LIN {X 0,Y 573.259,Z 217.079,A -85,B 0,C 180,E1 -2322.989,E2 -2322.989} C_VEL
LIN {X 0,Y 573.272,Z 217.08,A -85,B 0,C 180,E1 -2325.806,E2 -2325.806} C_VEL
LIN {X 0,Y 573.26,Z 217.081,A -85,B 0,C 180,E1 -2328.744,E2 -2328.744} C_VEL
LIN {X 0,Y 573.283,Z 217.076,A -85,B 0,C 180,E1 -2331.539,E2 -2331.539} C_VEL
LIN {X 0,Y 573.295,Z 217.075,A -85,B 0,C 180,E1 -2334.371,E2 -2334.371} C_VEL
LIN {X 0,Y 573.306,Z 217.073,A -85,B 0,C 180,E1 -2337.891,E2 -2337.891} C_VEL
LIN {X 0,Y 573.333,Z 217.07,A -85,B 0,C 180,E1 -2340.701,E2 -2340.701} C_VEL
LIN {X 0,Y 573.233,Z 217.085,A -85,B 0,C 180,E1 -2343.513,E2 -2343.513} C_VEL
LIN {X 0,Y 573.286,Z 217.078,A -85,B 0,C 180,E1 -2345.627,E2 -2345.627} C_VEL
LIN {X 0,Y 573.304,Z 217.075,A -85,B 0,C 180,E1 -2348.458,E2 -2348.458} C_VEL
LIN {X 0,Y 573.238,Z 217.083,A -85,B 0,C 180,E1 -2351.311,E2 -2351.311} C_VEL
LIN {X 0,Y 573.113,Z 217.279,A -85,B 0,C 180,E1 -2352.751,E2 -2352.751} C_VEL
LIN {X 0,Y 573.098,Z 219.875,A -85,B 0,C 180,E1 -2354.922,E2 -2354.922} C_VEL
LIN {X 0,Y 573.095,Z 222.437,A -85,B 0,C 180,E1 -2357.115,E2 -2357.115} C_VEL
LIN {X 0,Y 573.071,Z 224.992,A -85,B 0,C 180,E1 -2359.335,E2 -2359.335} C_VEL
LIN {X 0,Y 573.008,Z 227.552,A -85,B 0,C 180,E1 -2361.588,E2 -2361.588} C_VEL
LIN {X 0,Y 572.988,Z 230.552,A -85,B 0,C 180,E1 -2364.29,E2 -2364.29} C_VEL
LIN {X 0,Y 572.316,Z 231.276,A -85,B 0,C 180,E1 -2364.872,E2 -2364.872} C_VEL
LIN {X 0,Y 569.419,Z 232.626,A -85,B 0,C 180,E1 -2365.813,E2 -2365.813} C_VEL
LIN {X 0,Y 566.974,Z 233.725,A -85,B 0,C 180,E1 -2366.57,E2 -2366.57} C_VEL
LIN {X 0,Y 565.935,Z 234.507,A -85,B 0,C 180,E1 -2367.156,E2 -2367.156} C_VEL
LIN {X 0,Y 565.856,Z 234.734,A -85,B 0,C 180,E1 -2367.355,E2 -2367.355} C_VEL
LIN {X 0,Y 565.85,Z 237.623,A -85,B 0,C 180,E1 -2369.787,E2 -2369.787} C_VEL
LIN {X 0,Y 565.826,Z 240.978,A -85,B 0,C 180,E1 -2372.371,E2 -2372.371} C_VEL
LIN {X 0,Y 565.88,Z 243.683,A -85,B 0,C 180,E1 -2374.434,E2 -2374.434} C_VEL
LIN {X 0,Y 566.888,Z 251.451,A -85,B 0,C 180,E1 -2374.633,E2 -2374.633} C_VEL
LIN {X 0,Y 566.767,Z 263.644,A -85,B 0,C 180,E1 -2375.008,E2 -2375.008} C_VEL
LIN {X 0,Y 566.649,Z 274.804,A -85,B 0,C 180,E1 -2375.479,E2 -2375.479} C_VEL
LIN {X 0,Y 566.482,Z 285.658,A -85,B 0,C 180,E1 -2376.07,E2 -2376.07} C_VEL
LIN {X 0,Y 566.378,Z 296.002,A -85,B 0,C 180,E1 -2376.776,E2 -2376.776} C_VEL
LIN {X 0,Y 566.255,Z 306.666,A -85,B 0,C 180,E1 -2377.678,E2 -2377.678} C_VEL
LIN {X 0,Y 566.131,Z 316.26,A -85,B 0,C 180,E1 -2378.69,E2 -2378.69} C_VEL
LIN {X 0,Y 566.034,Z 323.764,A -85,B 0,C 180,E1 -2379.665,E2 -2379.665} C_VEL
LIN {X 0,Y 565.956,Z 330.595,A -85,B 0,C 180,E1 -2380.757,E2 -2380.757} C_VEL
LIN {X 0,Y 565.961,Z 335.973,A -85,B 0,C 180,E1 -2381.836,E2 -2381.836} C_VEL
LIN {X 0,Y 565.899,Z 340.744,A -85,B 0,C 180,E1 -2383.08,E2 -2383.08} C_VEL
LIN {X 0,Y 565.873,Z 343.485,A -85,B 0,C 180,E1 -2384.065,E2 -2384.065} C_VEL
LIN {X 0,Y 565.875,Z 345.441,A -85,B 0,C 180,E1 -2385.064,E2 -2385.064} C_VEL
LIN {X 0,Y 565.844,Z 346.619,A -85,B 0,C 180,E1 -2386.083,E2 -2386.083} C_VEL
LIN {X 0,Y 565.845,Z 346.99,A -85,B 0,C 180,E1 -2387.119,E2 -2387.119} C_VEL
LIN {X 0,Y 565.847,Z 346.5,A -85,B 0,C 180,E1 -2388.175,E2 -2388.175} C_VEL
LIN {X 0,Y 565.827,Z 345.077,A -85,B 0,C 180,E1 -2389.256,E2 -2389.256} C_VEL
LIN {X 0,Y 565.87,Z 342.663,A -85,B 0,C 180,E1 -2390.353,E2 -2390.353} C_VEL
LIN {X 0,Y 565.915,Z 338.608,A -85,B 0,C 180,E1 -2391.616,E2 -2391.616} C_VEL
LIN {X 0,Y 565.932,Z 334.259,A -85,B 0,C 180,E1 -2392.631,E2 -2392.631} C_VEL
LIN {X 0,Y 566.011,Z 327.802,A -85,B 0,C 180,E1 -2393.809,E2 -2393.809} C_VEL
LIN {X 0,Y 566.052,Z 320.425,A -85,B 0,C 180,E1 -2394.883,E2 -2394.883} C_VEL
LIN {X 0,Y 566.194,Z 311.453,A -85,B 0,C 180,E1 -2395.936,E2 -2395.936} C_VEL
LIN {X 0,Y 566.361,Z 301.081,A -85,B 0,C 180,E1 -2396.908,E2 -2396.908} C_VEL
LIN {X 0,Y 566.422,Z 289.815,A -85,B 0,C 180,E1 -2397.756,E2 -2397.756} C_VEL
LIN {X 0,Y 566.611,Z 278.018,A -85,B 0,C 180,E1 -2398.448,E2 -2398.448} C_VEL
LIN {X 0,Y 566.765,Z 265.989,A -85,B 0,C 180,E1 -2398.992,E2 -2398.992} C_VEL
LIN {X 0,Y 566.887,Z 253.367,A -85,B 0,C 180,E1 -2399.409,E2 -2399.409} C_VEL
LIN {X 0,Y 566.515,Z 247.713,A -85,B 0,C 180,E1 -2399.557,E2 -2399.557} C_VEL
LIN {X 0,Y 565.868,Z 243.662,A -85,B 0,C 180,E1 -2399.673,E2 -2399.673} C_VEL
LIN {X 0,Y 565.856,Z 239.773,A -85,B 0,C 180,E1 -2402.643,E2 -2402.643} C_VEL
LIN {X 0,Y 565.91,Z 236.681,A -85,B 0,C 180,E1 -2405.033,E2 -2405.033} C_VEL
LIN {X 0,Y 565.895,Z 233.927,A -85,B 0,C 180,E1 -2407.357,E2 -2407.357} C_VEL
LIN {X 0,Y 565.917,Z 230.496,A -85,B 0,C 180,E1 -2410.409,E2 -2410.409} C_VEL
LIN {X 0,Y 565.968,Z 226.89,A -85,B 0,C 180,E1 -2413.405,E2 -2413.405} C_VEL
LIN {X 0,Y 565.989,Z 223.532,A -85,B 0,C 180,E1 -2416.354,E2 -2416.354} C_VEL
LIN {X 0,Y 566.019,Z 220.045,A -85,B 0,C 180,E1 -2419.267,E2 -2419.267} C_VEL
LIN {X 0,Y 566.014,Z 218.352,A -85,B 0,C 180,E1 -2420.711,E2 -2420.711} C_VEL
LIN {X 0,Y 566.159,Z 217.965,A -85,B 0,C 180,E1 -2422.152,E2 -2422.152} C_VEL
LIN {X 0,Y 566.275,Z 217.949,A -85,B 0,C 180,E1 -2425.016,E2 -2425.016} C_VEL
LIN {X 0,Y 566.268,Z 217.95,A -85,B 0,C 180,E1 -2427.867,E2 -2427.867} C_VEL
LIN {X 0,Y 566.297,Z 217.949,A -85,B 0,C 180,E1 -2430.711,E2 -2430.711} C_VEL
LIN {X 0,Y 566.261,Z 217.952,A -85,B 0,C 180,E1 -2432.846,E2 -2432.846} C_VEL
LIN {X 0,Y 566.251,Z 217.952,A -85,B 0,C 180,E1 -2435.699,E2 -2435.699} C_VEL
LIN {X 0,Y 566.234,Z 217.953,A -85,B 0,C 180,E1 -2438.566,E2 -2438.566} C_VEL
LIN {X 0,Y 566.235,Z 217.955,A -85,B 0,C 180,E1 -2441.455,E2 -2441.455} C_VEL
LIN {X 0,Y 566.219,Z 217.955,A -85,B 0,C 180,E1 -2444.508,E2 -2444.508} C_VEL
LIN {X 0,Y 566.193,Z 217.961,A -85,B 0,C 180,E1 -2447.332,E2 -2447.332} C_VEL
LIN {X 0,Y 566.208,Z 217.957,A -85,B 0,C 180,E1 -2450.338,E2 -2450.338} C_VEL
LIN {X 0,Y 566.216,Z 217.957,A -85,B 0,C 180,E1 -2453.403,E2 -2453.403} C_VEL
LIN {X 0,Y 566.216,Z 217.958,A -85,B 0,C 180,E1 -2455.749,E2 -2455.749} C_VEL
LIN {X 0,Y 566.196,Z 217.96,A -85,B 0,C 180,E1 -2458.205,E2 -2458.205} C_VEL
LIN {X 0,Y 566.187,Z 217.959,A -85,B 0,C 180,E1 -2461.079,E2 -2461.079} C_VEL
LIN {X 0,Y 566.217,Z 217.956,A -85,B 0,C 180,E1 -2463.738,E2 -2463.738} C_VEL
LIN {X 0,Y 566.203,Z 217.959,A -85,B 0,C 180,E1 -2466.57,E2 -2466.57} C_VEL
LIN {X 0,Y 566.204,Z 217.958,A -85,B 0,C 180,E1 -2469.687,E2 -2469.687} C_VEL
LIN {X 0,Y 566.21,Z 217.957,A -85,B 0,C 180,E1 -2472.088,E2 -2472.088} C_VEL
LIN {X 0,Y 566.164,Z 217.963,A -85,B 0,C 180,E1 -2475.037,E2 -2475.037} C_VEL
LIN {X 0,Y 566.205,Z 217.957,A -85,B 0,C 180,E1 -2477.914,E2 -2477.914} C_VEL
LIN {X 0,Y 566.216,Z 217.958,A -85,B 0,C 180,E1 -2480.729,E2 -2480.729} C_VEL
LIN {X 0,Y 566.209,Z 217.956,A -85,B 0,C 180,E1 -2483.785,E2 -2483.785} C_VEL
LIN {X 0,Y 566.223,Z 217.955,A -85,B 0,C 180,E1 -2486.9,E2 -2486.9} C_VEL
LIN {X 0,Y 566.189,Z 217.959,A -85,B 0,C 180,E1 -2489.41,E2 -2489.41} C_VEL
LIN {X 0,Y 566.224,Z 217.955,A -85,B 0,C 180,E1 -2491.86,E2 -2491.86} C_VEL
LIN {X 0,Y 566.233,Z 217.956,A -85,B 0,C 180,E1 -2495.041,E2 -2495.041} C_VEL
LIN {X 0,Y 566.193,Z 217.959,A -85,B 0,C 180,E1 -2498.139,E2 -2498.139} C_VEL
LIN {X 0,Y 566.234,Z 217.954,A -85,B 0,C 180,E1 -2500.613,E2 -2500.613} C_VEL
LIN {X 0,Y 566.22,Z 217.958,A -85,B 0,C 180,E1 -2503.414,E2 -2503.414} C_VEL
LIN {X 0,Y 566.196,Z 217.958,A -85,B 0,C 180,E1 -2506.36,E2 -2506.36} C_VEL
LIN {X 0,Y 566.235,Z 217.953,A -85,B 0,C 180,E1 -2508.677,E2 -2508.677} C_VEL
LIN {X 0,Y 566.199,Z 217.959,A -85,B 0,C 180,E1 -2511.435,E2 -2511.435} C_VEL
LIN {X 0,Y 566.214,Z 217.956,A -85,B 0,C 180,E1 -2513.587,E2 -2513.587} C_VEL
LIN {X 0,Y 566.186,Z 217.96,A -85,B 0,C 180,E1 -2515.73,E2 -2515.73} C_VEL
LIN {X 0,Y 566.274,Z 217.95,A -85,B 0,C 180,E1 -2517.867,E2 -2517.867} C_VEL
LIN {X 0,Y 566.298,Z 217.945,A -85,B 0,C 180,E1 -2520.712,E2 -2520.712} C_VEL
LIN {X 0,Y 566.273,Z 217.949,A -85,B 0,C 180,E1 -2522.847,E2 -2522.847} C_VEL
LIN {X 0,Y 566.259,Z 217.951,A -85,B 0,C 180,E1 -2525.699,E2 -2525.699} C_VEL
LIN {X 0,Y 566.209,Z 217.958,A -85,B 0,C 180,E1 -2528.567,E2 -2528.567} C_VEL
LIN {X 0,Y 566.247,Z 217.952,A -85,B 0,C 180,E1 -2531.455,E2 -2531.455} C_VEL
LIN {X 0,Y 566.235,Z 217.955,A -85,B 0,C 180,E1 -2534.506,E2 -2534.506} C_VEL
LIN {X 0,Y 566.208,Z 217.957,A -85,B 0,C 180,E1 -2537.332,E2 -2537.332} C_VEL
LIN {X 0,Y 566.212,Z 217.959,A -85,B 0,C 180,E1 -2540.338,E2 -2540.338} C_VEL
LIN {X 0,Y 566.175,Z 217.961,A -85,B 0,C 180,E1 -2543.282,E2 -2543.282} C_VEL
LIN {X 0,Y 566.207,Z 217.957,A -85,B 0,C 180,E1 -2545.75,E2 -2545.75} C_VEL
LIN {X 0,Y 566.209,Z 217.957,A -85,B 0,C 180,E1 -2548.203,E2 -2548.203} C_VEL
LIN {X 0,Y 566.191,Z 217.962,A -85,B 0,C 180,E1 -2551.076,E2 -2551.076} C_VEL
LIN {X 0,Y 566.203,Z 217.958,A -85,B 0,C 180,E1 -2553.732,E2 -2553.732} C_VEL
LIN {X 0,Y 566.205,Z 217.957,A -85,B 0,C 180,E1 -2556.57,E2 -2556.57} C_VEL
LIN {X 0,Y 566.22,Z 217.955,A -85,B 0,C 180,E1 -2559.686,E2 -2559.686} C_VEL
LIN {X 0,Y 566.207,Z 217.959,A -85,B 0,C 180,E1 -2562.917,E2 -2562.917} C_VEL
LIN {X 0,Y 566.2,Z 217.957,A -85,B 0,C 180,E1 -2566.049,E2 -2566.049} C_VEL
LIN {X 0,Y 566.209,Z 217.958,A -85,B 0,C 180,E1 -2569.215,E2 -2569.215} C_VEL
LIN {X 0,Y 566.19,Z 217.96,A -85,B 0,C 180,E1 -2571.637,E2 -2571.637} C_VEL
LIN {X 0,Y 566.227,Z 218.124,A -85,B 0,C 180,E1 -2573.043,E2 -2573.043} C_VEL
LIN {X 0,Y 566.797,Z 221.916,A -85,B 0,C 180,E1 -2574.354,E2 -2574.354} C_VEL
LIN {X 0,Y 566.804,Z 228.677,A -85,B 0,C 180,E1 -2576.557,E2 -2576.557} C_VEL
LIN {X 0,Y 566.614,Z 237.802,A -85,B 0,C 180,E1 -2579.433,E2 -2579.433} C_VEL
LIN {X 0,Y 566.507,Z 247.07,A -85,B 0,C 180,E1 -2582.275,E2 -2582.275} C_VEL
LIN {X 0,Y 566.417,Z 256.337,A -85,B 0,C 180,E1 -2585.047,E2 -2585.047} C_VEL
LIN {X 0,Y 566.324,Z 266.928,A -85,B 0,C 180,E1 -2588.142,E2 -2588.142} C_VEL
LIN {X 0,Y 566.187,Z 277.519,A -85,B 0,C 180,E1 -2591.171,E2 -2591.171} C_VEL
LIN {X 0,Y 566.114,Z 288.11,A -85,B 0,C 180,E1 -2594.15,E2 -2594.15} C_VEL
LIN {X 0,Y 566.003,Z 298.702,A -85,B 0,C 180,E1 -2597.085,E2 -2597.085} C_VEL
LIN {X 0,Y 566.013,Z 299.529,A -85,B 0,C 180,E1 -2597.313,E2 -2597.313} C_VEL
LIN {X 0,Y 566.933,Z 306.354,A -85,B 0,C 180,E1 -2597.47,E2 -2597.47} C_VEL
LIN {X 0,Y 566.841,Z 318.486,A -85,B 0,C 180,E1 -2597.786,E2 -2597.786} C_VEL
LIN {X 0,Y 566.688,Z 330.312,A -85,B 0,C 180,E1 -2598.228,E2 -2598.228} C_VEL
LIN {X 0,Y 566.534,Z 342.974,A -85,B 0,C 180,E1 -2598.868,E2 -2598.868} C_VEL
LIN {X 0,Y 566.454,Z 354.742,A -85,B 0,C 180,E1 -2599.636,E2 -2599.636} C_VEL
LIN {X 0,Y 566.302,Z 363.643,A -85,B 0,C 180,E1 -2600.355,E2 -2600.355} C_VEL
LIN {X 0,Y 566.162,Z 372.784,A -85,B 0,C 180,E1 -2601.253,E2 -2601.253} C_VEL
LIN {X 0,Y 566.081,Z 381.688,A -85,B 0,C 180,E1 -2602.33,E2 -2602.33} C_VEL
LIN {X 0,Y 565.969,Z 388.953,A -85,B 0,C 180,E1 -2603.422,E2 -2603.422} C_VEL
LIN {X 0,Y 566.004,Z 393.678,A -85,B 0,C 180,E1 -2604.299,E2 -2604.299} C_VEL
LIN {X 0,Y 565.933,Z 398.37,A -85,B 0,C 180,E1 -2605.37,E2 -2605.37} C_VEL
LIN {X 0,Y 565.927,Z 401.955,A -85,B 0,C 180,E1 -2606.44,E2 -2606.44} C_VEL
LIN {X 0,Y 565.878,Z 403.808,A -85,B 0,C 180,E1 -2607.152,E2 -2607.152} C_VEL
LIN {X 0,Y 565.841,Z 405.199,A -85,B 0,C 180,E1 -2607.864,E2 -2607.864} C_VEL
LIN {X 0,Y 565.841,Z 406.784,A -85,B 0,C 180,E1 -2609.288,E2 -2609.288} C_VEL
LIN {X 0,Y 565.839,Z 407,A -85,B 0,C 180,E1 -2610,E2 -2610} C_VEL
LIN {X 0,Y 565.846,Z 406.186,A -85,B 0,C 180,E1 -2611.423,E2 -2611.423} C_VEL
LIN {X 0,Y 565.841,Z 405.202,A -85,B 0,C 180,E1 -2612.135,E2 -2612.135} C_VEL
LIN {X 0,Y 565.878,Z 403.811,A -85,B 0,C 180,E1 -2612.847,E2 -2612.847} C_VEL
LIN {X 0,Y 565.926,Z 400.897,A -85,B 0,C 180,E1 -2613.916,E2 -2613.916} C_VEL
LIN {X 0,Y 565.878,Z 396.951,A -85,B 0,C 180,E1 -2614.987,E2 -2614.987} C_VEL
LIN {X 0,Y 566.002,Z 391.869,A -85,B 0,C 180,E1 -2616.058,E2 -2616.058} C_VEL
LIN {X 0,Y 566.041,Z 385.473,A -85,B 0,C 180,E1 -2617.132,E2 -2617.132} C_VEL
LIN {X 0,Y 566.134,Z 377.482,A -85,B 0,C 180,E1 -2618.207,E2 -2618.207} C_VEL
LIN {X 0,Y 566.229,Z 369.341,A -85,B 0,C 180,E1 -2619.105,E2 -2619.105} C_VEL
LIN {X 0,Y 566.349,Z 359.408,A -85,B 0,C 180,E1 -2620.004,E2 -2620.004} C_VEL
LIN {X 0,Y 566.503,Z 348.324,A -85,B 0,C 180,E1 -2620.805,E2 -2620.805} C_VEL
LIN {X 0,Y 566.609,Z 335.96,A -85,B 0,C 180,E1 -2621.509,E2 -2621.509} C_VEL
LIN {X 0,Y 566.773,Z 323.78,A -85,B 0,C 180,E1 -2622.032,E2 -2622.032} C_VEL
LIN {X 0,Y 566.915,Z 311.283,A -85,B 0,C 180,E1 -2622.416,E2 -2622.416} C_VEL
LIN {X 0,Y 566.731,Z 304.111,A -85,B 0,C 180,E1 -2622.579,E2 -2622.579} C_VEL
LIN {X 0,Y 566.012,Z 299.532,A -85,B 0,C 180,E1 -2622.686,E2 -2622.686} C_VEL
LIN {X 0,Y 566.088,Z 289.437,A -85,B 0,C 180,E1 -2625.481,E2 -2625.481} C_VEL
LIN {X 0,Y 566.167,Z 278.846,A -85,B 0,C 180,E1 -2628.453,E2 -2628.453} C_VEL
LIN {X 0,Y 566.24,Z 269.579,A -85,B 0,C 180,E1 -2631.096,E2 -2631.096} C_VEL
LIN {X 0,Y 566.364,Z 260.312,A -85,B 0,C 180,E1 -2633.784,E2 -2633.784} C_VEL
LIN {X 0,Y 566.458,Z 250.445,A -85,B 0,C 180,E1 -2636.708,E2 -2636.708} C_VEL
LIN {X 0,Y 566.548,Z 241.777,A -85,B 0,C 180,E1 -2639.34,E2 -2639.34} C_VEL
LIN {X 0,Y 566.7,Z 232.51,A -85,B 0,C 180,E1 -2642.226,E2 -2642.226} C_VEL
LIN {X 0,Y 566.837,Z 224.566,A -85,B 0,C 180,E1 -2644.773,E2 -2644.773} C_VEL
LIN {X 0,Y 566.577,Z 220.063,A -85,B 0,C 180,E1 -2646.265,E2 -2646.265} C_VEL
LIN {X 0,Y 566.236,Z 217.957,A -85,B 0,C 180,E1 -2647.011,E2 -2647.011} C_VEL
LIN {X 0,Y 566.214,Z 217.958,A -85,B 0,C 180,E1 -2649.685,E2 -2649.685} C_VEL
LIN {X 0,Y 566.203,Z 217.959,A -85,B 0,C 180,E1 -2652.916,E2 -2652.916} C_VEL
LIN {X 0,Y 566.199,Z 217.958,A -85,B 0,C 180,E1 -2656.048,E2 -2656.048} C_VEL
LIN {X 0,Y 566.213,Z 217.958,A -85,B 0,C 180,E1 -2658.863,E2 -2658.863} C_VEL
LIN {X 0,Y 566.191,Z 217.961,A -85,B 0,C 180,E1 -2661.636,E2 -2661.636} C_VEL
LIN {X 0,Y 566.163,Z 217.964,A -85,B 0,C 180,E1 -2664.307,E2 -2664.307} C_VEL
LIN {X 0,Y 566.219,Z 217.958,A -85,B 0,C 180,E1 -2666.897,E2 -2666.897} C_VEL
LIN {X 0,Y 566.184,Z 217.961,A -85,B 0,C 180,E1 -2669.407,E2 -2669.407} C_VEL
LIN {X 0,Y 566.228,Z 217.955,A -85,B 0,C 180,E1 -2671.857,E2 -2671.857} C_VEL
LIN {X 0,Y 566.226,Z 217.958,A -85,B 0,C 180,E1 -2674.251,E2 -2674.251} C_VEL
LIN {X 0,Y 566.191,Z 217.96,A -85,B 0,C 180,E1 -2676.713,E2 -2676.713} C_VEL
LIN {X 0,Y 566.219,Z 217.957,A -85,B 0,C 180,E1 -2679.662,E2 -2679.662} C_VEL
LIN {X 0,Y 566.199,Z 217.961,A -85,B 0,C 180,E1 -2682.667,E2 -2682.667} C_VEL
LIN {X 0,Y 566.232,Z 217.956,A -85,B 0,C 180,E1 -2685.626,E2 -2685.626} C_VEL
LIN {X 0,Y 566.232,Z 217.956,A -85,B 0,C 180,E1 -2688.674,E2 -2688.674} C_VEL
LIN {X 0,Y 566.227,Z 217.954,A -85,B 0,C 180,E1 -2691.433,E2 -2691.433} C_VEL
LIN {X 0,Y 566.262,Z 217.952,A -85,B 0,C 180,E1 -2694.301,E2 -2694.301} C_VEL
LIN {X 0,Y 566.277,Z 217.949,A -85,B 0,C 180,E1 -2697.865,E2 -2697.865} C_VEL
LIN {X 0,Y 566.303,Z 217.946,A -85,B 0,C 180,E1 -2700.71,E2 -2700.71} C_VEL
LIN {X 0,Y 566.271,Z 217.95,A -85,B 0,C 180,E1 -2702.844,E2 -2702.844} C_VEL
LIN {X 0,Y 566.255,Z 217.953,A -85,B 0,C 180,E1 -2705.697,E2 -2705.697} C_VEL
LIN {X 0,Y 566.245,Z 217.955,A -85,B 0,C 180,E1 -2708.564,E2 -2708.564} C_VEL
LIN {X 0,Y 566.184,Z 217.962,A -85,B 0,C 180,E1 -2711.454,E2 -2711.454} C_VEL
LIN {X 0,Y 566.053,Z 218.193,A -85,B 0,C 180,E1 -2712.912,E2 -2712.912} C_VEL
LIN {X 0,Y 566.033,Z 220.785,A -85,B 0,C 180,E1 -2715.113,E2 -2715.113} C_VEL
LIN {X 0,Y 566.023,Z 223.36,A -85,B 0,C 180,E1 -2717.336,E2 -2717.336} C_VEL
LIN {X 0,Y 566,Z 225.934,A -85,B 0,C 180,E1 -2719.587,E2 -2719.587} C_VEL
LIN {X 0,Y 565.924,Z 229.364,A -85,B 0,C 180,E1 -2722.641,E2 -2722.641} C_VEL
LIN {X 0,Y 565.908,Z 231.982,A -85,B 0,C 180,E1 -2724.975,E2 -2724.975} C_VEL
LIN {X 0,Y 565.856,Z 234.734,A -85,B 0,C 180,E1 -2727.355,E2 -2727.355} C_VEL
LIN {X 0,Y 565.201,Z 235.469,A -85,B 0,C 180,E1 -2727.945,E2 -2727.945} C_VEL
LIN {X 0,Y 562.334,Z 236.795,A -85,B 0,C 180,E1 -2728.9,E2 -2728.9} C_VEL
LIN {X 0,Y 559.895,Z 237.861,A -85,B 0,C 180,E1 -2729.669,E2 -2729.669} C_VEL
LIN {X 0,Y 558.838,Z 238.619,A -85,B 0,C 180,E1 -2730.264,E2 -2730.264} C_VEL
LIN {X 0,Y 558.748,Z 238.855,A -85,B 0,C 180,E1 -2730.465,E2 -2730.465} C_VEL
LIN {X 0,Y 558.743,Z 242.815,A -85,B 0,C 180,E1 -2733.601,E2 -2733.601} C_VEL
LIN {X 0,Y 558.777,Z 243.681,A -85,B 0,C 180,E1 -2734.269,E2 -2734.269} C_VEL
LIN {X 0,Y 559.951,Z 251.642,A -85,B 0,C 180,E1 -2734.482,E2 -2734.482} C_VEL
LIN {X 0,Y 559.812,Z 264.517,A -85,B 0,C 180,E1 -2734.888,E2 -2734.888} C_VEL
LIN {X 0,Y 559.683,Z 275.562,A -85,B 0,C 180,E1 -2735.371,E2 -2735.371} C_VEL
LIN {X 0,Y 559.456,Z 287.715,A -85,B 0,C 180,E1 -2736.062,E2 -2736.062} C_VEL
LIN {X 0,Y 559.344,Z 298.439,A -85,B 0,C 180,E1 -2736.836,E2 -2736.836} C_VEL
LIN {X 0,Y 559.199,Z 307.611,A -85,B 0,C 180,E1 -2737.649,E2 -2737.649} C_VEL
LIN {X 0,Y 559.075,Z 316.688,A -85,B 0,C 180,E1 -2738.636,E2 -2738.636} C_VEL
LIN {X 0,Y 558.98,Z 324.274,A -85,B 0,C 180,E1 -2739.646,E2 -2739.646} C_VEL
LIN {X 0,Y 558.884,Z 331.467,A -85,B 0,C 180,E1 -2740.834,E2 -2740.834} C_VEL
LIN {X 0,Y 558.84,Z 337.363,A -85,B 0,C 180,E1 -2742.1,E2 -2742.1} C_VEL
LIN {X 0,Y 558.808,Z 341.137,A -85,B 0,C 180,E1 -2743.16,E2 -2743.16} C_VEL
LIN {X 0,Y 558.785,Z 343.897,A -85,B 0,C 180,E1 -2744.201,E2 -2744.201} C_VEL
LIN {X 0,Y 558.782,Z 345.728,A -85,B 0,C 180,E1 -2745.225,E2 -2745.225} C_VEL
LIN {X 0,Y 558.751,Z 346.723,A -85,B 0,C 180,E1 -2746.229,E2 -2746.229} C_VEL
LIN {X 0,Y 558.741,Z 346.969,A -85,B 0,C 180,E1 -2747.218,E2 -2747.218} C_VEL
LIN {X 0,Y 558.751,Z 346.497,A -85,B 0,C 180,E1 -2748.193,E2 -2748.193} C_VEL
LIN {X 0,Y 558.746,Z 345.282,A -85,B 0,C 180,E1 -2749.152,E2 -2749.152} C_VEL
LIN {X 0,Y 558.776,Z 342.198,A -85,B 0,C 180,E1 -2750.569,E2 -2750.569} C_VEL
LIN {X 0,Y 558.83,Z 338.904,A -85,B 0,C 180,E1 -2751.596,E2 -2751.596} C_VEL
LIN {X 0,Y 558.85,Z 333.427,A -85,B 0,C 180,E1 -2752.87,E2 -2752.87} C_VEL
LIN {X 0,Y 558.948,Z 327.165,A -85,B 0,C 180,E1 -2753.998,E2 -2753.998} C_VEL
LIN {X 0,Y 559.004,Z 319.486,A -85,B 0,C 180,E1 -2755.108,E2 -2755.108} C_VEL
LIN {X 0,Y 559.164,Z 311.464,A -85,B 0,C 180,E1 -2756.048,E2 -2756.048} C_VEL
LIN {X 0,Y 559.325,Z 301.759,A -85,B 0,C 180,E1 -2756.975,E2 -2756.975} C_VEL
LIN {X 0,Y 559.422,Z 290.616,A -85,B 0,C 180,E1 -2757.836,E2 -2757.836} C_VEL
LIN {X 0,Y 559.609,Z 279.715,A -85,B 0,C 180,E1 -2758.504,E2 -2758.504} C_VEL
LIN {X 0,Y 559.797,Z 267.709,A -85,B 0,C 180,E1 -2759.073,E2 -2759.073} C_VEL
LIN {X 0,Y 559.942,Z 254.682,A -85,B 0,C 180,E1 -2759.526,E2 -2759.526} C_VEL
LIN {X 0,Y 559.725,Z 249.414,A -85,B 0,C 180,E1 -2759.67,E2 -2759.67} C_VEL
LIN {X 0,Y 558.761,Z 243.678,A -85,B 0,C 180,E1 -2759.824,E2 -2759.824} C_VEL
LIN {X 0,Y 558.747,Z 240.52,A -85,B 0,C 180,E1 -2762.265,E2 -2762.265} C_VEL
LIN {X 0,Y 558.805,Z 237.329,A -85,B 0,C 180,E1 -2764.89,E2 -2764.89} C_VEL
LIN {X 0,Y 558.829,Z 234.84,A -85,B 0,C 180,E1 -2767.054,E2 -2767.054} C_VEL
LIN {X 0,Y 558.849,Z 231.356,A -85,B 0,C 180,E1 -2770.151,E2 -2770.151} C_VEL
LIN {X 0,Y 558.887,Z 227.739,A -85,B 0,C 180,E1 -2773.189,E2 -2773.189} C_VEL
LIN {X 0,Y 558.938,Z 224.335,A -85,B 0,C 180,E1 -2776.179,E2 -2776.179} C_VEL
LIN {X 0,Y 558.967,Z 220.846,A -85,B 0,C 180,E1 -2779.129,E2 -2779.129} C_VEL
LIN {X 0,Y 558.938,Z 219.139,A -85,B 0,C 180,E1 -2780.593,E2 -2780.593} C_VEL
LIN {X 0,Y 559.104,Z 218.844,A -85,B 0,C 180,E1 -2782.053,E2 -2782.053} C_VEL
LIN {X 0,Y 559.219,Z 218.827,A -85,B 0,C 180,E1 -2784.23,E2 -2784.23} C_VEL
LIN {X 0,Y 559.226,Z 218.83,A -85,B 0,C 180,E1 -2787.119,E2 -2787.119} C_VEL
LIN {X 0,Y 559.244,Z 218.824,A -85,B 0,C 180,E1 -2790,E2 -2790} C_VEL
LIN {X 0,Y 559.227,Z 218.828,A -85,B 0,C 180,E1 -2792.882,E2 -2792.882} C_VEL
LIN {X 0,Y 559.219,Z 218.827,A -85,B 0,C 180,E1 -2795.771,E2 -2795.771} C_VEL
LIN {X 0,Y 559.188,Z 218.832,A -85,B 0,C 180,E1 -2798.675,E2 -2798.675} C_VEL
LIN {X 0,Y 559.194,Z 218.831,A -85,B 0,C 180,E1 -2801.601,E2 -2801.601} C_VEL
LIN {X 0,Y 559.183,Z 218.832,A -85,B 0,C 180,E1 -2804.596,E2 -2804.596} C_VEL
LIN {X 0,Y 559.152,Z 218.836,A -85,B 0,C 180,E1 -2807.557,E2 -2807.557} C_VEL
LIN {X 0,Y 559.174,Z 218.834,A -85,B 0,C 180,E1 -2810.605,E2 -2810.605} C_VEL
LIN {X 0,Y 559.153,Z 218.835,A -85,B 0,C 180,E1 -2813.717,E2 -2813.717} C_VEL
LIN {X 0,Y 559.188,Z 218.831,A -85,B 0,C 180,E1 -2816.097,E2 -2816.097} C_VEL
LIN {X 0,Y 559.154,Z 218.836,A -85,B 0,C 180,E1 -2818.53,E2 -2818.53} C_VEL
LIN {X 0,Y 559.142,Z 218.838,A -85,B 0,C 180,E1 -2821.276,E2 -2821.276} C_VEL
LIN {X 0,Y 559.166,Z 218.836,A -85,B 0,C 180,E1 -2823.952,E2 -2823.952} C_VEL
LIN {X 0,Y 559.156,Z 218.838,A -85,B 0,C 180,E1 -2826.45,E2 -2826.45} C_VEL
LIN {X 0,Y 559.168,Z 218.835,A -85,B 0,C 180,E1 -2828.935,E2 -2828.935} C_VEL
LIN {X 0,Y 559.188,Z 218.831,A -85,B 0,C 180,E1 -2831.768,E2 -2831.768} C_VEL
LIN {X 0,Y 559.131,Z 218.841,A -85,B 0,C 180,E1 -2834.74,E2 -2834.74} C_VEL
LIN {X 0,Y 559.155,Z 218.837,A -85,B 0,C 180,E1 -2837.258,E2 -2837.258} C_VEL
LIN {X 0,Y 559.179,Z 218.832,A -85,B 0,C 180,E1 -2840.137,E2 -2840.137} C_VEL
LIN {X 0,Y 559.14,Z 218.839,A -85,B 0,C 180,E1 -2842.894,E2 -2842.894} C_VEL
LIN {X 0,Y 559.17,Z 218.833,A -85,B 0,C 180,E1 -2846.051,E2 -2846.051} C_VEL
LIN {X 0,Y 559.162,Z 218.837,A -85,B 0,C 180,E1 -2848.983,E2 -2848.983} C_VEL
LIN {X 0,Y 559.167,Z 218.836,A -85,B 0,C 180,E1 -2851.62,E2 -2851.62} C_VEL
LIN {X 0,Y 559.172,Z 218.834,A -85,B 0,C 180,E1 -2854.703,E2 -2854.703} C_VEL
LIN {X 0,Y 559.129,Z 218.839,A -85,B 0,C 180,E1 -2857.069,E2 -2857.069} C_VEL
LIN {X 0,Y 559.177,Z 218.832,A -85,B 0,C 180,E1 -2859.397,E2 -2859.397} C_VEL
LIN {X 0,Y 559.151,Z 218.836,A -85,B 0,C 180,E1 -2861.687,E2 -2861.687} C_VEL
LIN {X 0,Y 559.169,Z 218.834,A -85,B 0,C 180,E1 -2863.949,E2 -2863.949} C_VEL
LIN {X 0,Y 559.171,Z 218.834,A -85,B 0,C 180,E1 -2866.186,E2 -2866.186} C_VEL
LIN {X 0,Y 559.196,Z 218.832,A -85,B 0,C 180,E1 -2869.135,E2 -2869.135} C_VEL
LIN {X 0,Y 559.191,Z 218.831,A -85,B 0,C 180,E1 -2872.055,E2 -2872.055} C_VEL
LIN {X 0,Y 559.254,Z 218.823,A -85,B 0,C 180,E1 -2874.955,E2 -2874.955} C_VEL
LIN {X 0,Y 559.246,Z 218.825,A -85,B 0,C 180,E1 -2877.841,E2 -2877.841} C_VEL
LIN {X 0,Y 559.269,Z 218.82,A -85,B 0,C 180,E1 -2880.721,E2 -2880.721} C_VEL
LIN {X 0,Y 559.239,Z 218.824,A -85,B 0,C 180,E1 -2882.883,E2 -2882.883} C_VEL
LIN {X 0,Y 559.227,Z 218.828,A -85,B 0,C 180,E1 -2885.771,E2 -2885.771} C_VEL
LIN {X 0,Y 559.174,Z 218.833,A -85,B 0,C 180,E1 -2888.676,E2 -2888.676} C_VEL
LIN {X 0,Y 559.21,Z 218.829,A -85,B 0,C 180,E1 -2891.601,E2 -2891.601} C_VEL
LIN {X 0,Y 559.205,Z 218.83,A -85,B 0,C 180,E1 -2894.596,E2 -2894.596} C_VEL
LIN {X 0,Y 559.167,Z 218.835,A -85,B 0,C 180,E1 -2897.558,E2 -2897.558} C_VEL
LIN {X 0,Y 559.171,Z 218.834,A -85,B 0,C 180,E1 -2899.838,E2 -2899.838} C_VEL
LIN {X 0,Y 559.146,Z 218.836,A -85,B 0,C 180,E1 -2902.154,E2 -2902.154} C_VEL
LIN {X 0,Y 559.144,Z 218.839,A -85,B 0,C 180,E1 -2905.179,E2 -2905.179} C_VEL
LIN {X 0,Y 559.187,Z 218.832,A -85,B 0,C 180,E1 -2907.713,E2 -2907.713} C_VEL
LIN {X 0,Y 559.153,Z 218.835,A -85,B 0,C 180,E1 -2910.184,E2 -2910.184} C_VEL
LIN {X 0,Y 559.158,Z 218.835,A -85,B 0,C 180,E1 -2912.716,E2 -2912.716} C_VEL
LIN {X 0,Y 559.134,Z 218.838,A -85,B 0,C 180,E1 -2915.325,E2 -2915.325} C_VEL
LIN {X 0,Y 559.139,Z 218.839,A -85,B 0,C 180,E1 -2918.018,E2 -2918.018} C_VEL
LIN {X 0,Y 559.161,Z 218.836,A -85,B 0,C 180,E1 -2920.813,E2 -2920.813} C_VEL
LIN {X 0,Y 559.146,Z 218.836,A -85,B 0,C 180,E1 -2923.734,E2 -2923.734} C_VEL
LIN {X 0,Y 559.151,Z 218.836,A -85,B 0,C 180,E1 -2926.804,E2 -2926.804} C_VEL
LIN {X 0,Y 559.161,Z 218.836,A -85,B 0,C 180,E1 -2929.188,E2 -2929.188} C_VEL
LIN {X 0,Y 559.136,Z 218.838,A -85,B 0,C 180,E1 -2931.982,E2 -2931.982} C_VEL
LIN {X 0,Y 559.184,Z 219.009,A -85,B 0,C 180,E1 -2932.797,E2 -2932.797} C_VEL
LIN {X 0,Y 559.848,Z 223.251,A -85,B 0,C 180,E1 -2934.287,E2 -2934.287} C_VEL
LIN {X 0,Y 559.851,Z 229.859,A -85,B 0,C 180,E1 -2936.472,E2 -2936.472} C_VEL
LIN {X 0,Y 559.64,Z 239.126,A -85,B 0,C 180,E1 -2939.429,E2 -2939.429} C_VEL
LIN {X 0,Y 559.519,Z 248.394,A -85,B 0,C 180,E1 -2942.306,E2 -2942.306} C_VEL
LIN {X 0,Y 559.396,Z 257.749,A -85,B 0,C 180,E1 -2945.136,E2 -2945.136} C_VEL
LIN {X 0,Y 559.293,Z 266.928,A -85,B 0,C 180,E1 -2947.853,E2 -2947.853} C_VEL
LIN {X 0,Y 559.147,Z 277.519,A -85,B 0,C 180,E1 -2950.925,E2 -2950.925} C_VEL
LIN {X 0,Y 559.056,Z 286.786,A -85,B 0,C 180,E1 -2953.569,E2 -2953.569} C_VEL
LIN {X 0,Y 558.961,Z 297.378,A -85,B 0,C 180,E1 -2956.549,E2 -2956.549} C_VEL
LIN {X 0,Y 558.939,Z 299.529,A -85,B 0,C 180,E1 -2957.15,E2 -2957.15} C_VEL
LIN {X 0,Y 560.018,Z 307.494,A -85,B 0,C 180,E1 -2957.336,E2 -2957.336} C_VEL
LIN {X 0,Y 559.899,Z 319.868,A -85,B 0,C 180,E1 -2957.679,E2 -2957.679} C_VEL
LIN {X 0,Y 559.712,Z 332.275,A -85,B 0,C 180,E1 -2958.17,E2 -2958.17} C_VEL
LIN {X 0,Y 559.557,Z 343.761,A -85,B 0,C 180,E1 -2958.773,E2 -2958.773} C_VEL
LIN {X 0,Y 559.451,Z 354.742,A -85,B 0,C 180,E1 -2959.504,E2 -2959.504} C_VEL
LIN {X 0,Y 559.245,Z 365.597,A -85,B 0,C 180,E1 -2960.415,E2 -2960.415} C_VEL
LIN {X 0,Y 559.123,Z 374.41,A -85,B 0,C 180,E1 -2961.324,E2 -2961.324} C_VEL
LIN {X 0,Y 558.997,Z 382.998,A -85,B 0,C 180,E1 -2962.414,E2 -2962.414} C_VEL
LIN {X 0,Y 558.886,Z 390.689,A -85,B 0,C 180,E1 -2963.649,E2 -2963.649} C_VEL
LIN {X 0,Y 558.869,Z 395.364,A -85,B 0,C 180,E1 -2964.588,E2 -2964.588} C_VEL
LIN {X 0,Y 558.869,Z 399.676,A -85,B 0,C 180,E1 -2965.672,E2 -2965.672} C_VEL
LIN {X 0,Y 558.836,Z 401.956,A -85,B 0,C 180,E1 -2966.394,E2 -2966.394} C_VEL
LIN {X 0,Y 558.799,Z 403.808,A -85,B 0,C 180,E1 -2967.116,E2 -2967.116} C_VEL
LIN {X 0,Y 558.747,Z 405.199,A -85,B 0,C 180,E1 -2967.837,E2 -2967.837} C_VEL
LIN {X 0,Y 558.741,Z 406.784,A -85,B 0,C 180,E1 -2969.279,E2 -2969.279} C_VEL
LIN {X 0,Y 558.74,Z 407,A -85,B 0,C 180,E1 -2970,E2 -2970} C_VEL
LIN {X 0,Y 558.745,Z 406.186,A -85,B 0,C 180,E1 -2971.441,E2 -2971.441} C_VEL
LIN {X 0,Y 558.747,Z 405.201,A -85,B 0,C 180,E1 -2972.162,E2 -2972.162} C_VEL
LIN {X 0,Y 558.799,Z 403.811,A -85,B 0,C 180,E1 -2972.883,E2 -2972.883} C_VEL
LIN {X 0,Y 558.844,Z 400.897,A -85,B 0,C 180,E1 -2973.966,E2 -2973.966} C_VEL
LIN {X 0,Y 558.798,Z 396.951,A -85,B 0,C 180,E1 -2975.05,E2 -2975.05} C_VEL
LIN {X 0,Y 558.922,Z 391.869,A -85,B 0,C 180,E1 -2976.135,E2 -2976.135} C_VEL
LIN {X 0,Y 558.978,Z 385.472,A -85,B 0,C 180,E1 -2977.222,E2 -2977.222} C_VEL
LIN {X 0,Y 559.099,Z 377.482,A -85,B 0,C 180,E1 -2978.311,E2 -2978.311} C_VEL
LIN {X 0,Y 559.195,Z 369.341,A -85,B 0,C 180,E1 -2979.221,E2 -2979.221} C_VEL
LIN {X 0,Y 559.35,Z 359.407,A -85,B 0,C 180,E1 -2980.131,E2 -2980.131} C_VEL
LIN {X 0,Y 559.506,Z 348.429,A -85,B 0,C 180,E1 -2980.935,E2 -2980.935} C_VEL
LIN {X 0,Y 559.636,Z 336.832,A -85,B 0,C 180,E1 -2981.609,E2 -2981.609} C_VEL
LIN {X 0,Y 559.798,Z 324.999,A -85,B 0,C 180,E1 -2982.139,E2 -2982.139} C_VEL
LIN {X 0,Y 559.952,Z 312.196,A -85,B 0,C 180,E1 -2982.549,E2 -2982.549} C_VEL
LIN {X 0,Y 559.815,Z 304.968,A -85,B 0,C 180,E1 -2982.72,E2 -2982.72} C_VEL
LIN {X 0,Y 558.938,Z 299.532,A -85,B 0,C 180,E1 -2982.85,E2 -2982.85} C_VEL
LIN {X 0,Y 559.053,Z 289.437,A -85,B 0,C 180,E1 -2985.681,E2 -2985.681} C_VEL
LIN {X 0,Y 559.134,Z 278.846,A -85,B 0,C 180,E1 -2988.694,E2 -2988.694} C_VEL
LIN {X 0,Y 559.224,Z 268.92,A -85,B 0,C 180,E1 -2991.566,E2 -2991.566} C_VEL
LIN {X 0,Y 559.376,Z 258.988,A -85,B 0,C 180,E1 -2994.494,E2 -2994.494} C_VEL
LIN {X 0,Y 559.495,Z 249.72,A -85,B 0,C 180,E1 -2997.289,E2 -2997.289} C_VEL
LIN {X 0,Y 559.64,Z 240.453,A -85,B 0,C 180,E1 -3000.153,E2 -3000.153} C_VEL
LIN {X 0,Y 559.792,Z 231.187,A -85,B 0,C 180,E1 -3003.101,E2 -3003.101} C_VEL
LIN {X 0,Y 559.866,Z 223.183,A -85,B 0,C 180,E1 -3005.711,E2 -3005.711} C_VEL
LIN {X 0,Y 559.172,Z 218.837,A -85,B 0,C 180,E1 -3007.301,E2 -3007.301} C_VEL
LIN {X 0,Y 559.161,Z 218.836,A -85,B 0,C 180,E1 -3009.941,E2 -3009.941} C_VEL
LIN {X 0,Y 559.159,Z 218.837,A -85,B 0,C 180,E1 -3012.743,E2 -3012.743} C_VEL
LIN {X 0,Y 559.154,Z 218.837,A -85,B 0,C 180,E1 -3015.76,E2 -3015.76} C_VEL
LIN {X 0,Y 559.193,Z 218.832,A -85,B 0,C 180,E1 -3018.232,E2 -3018.232} C_VEL
LIN {X 0,Y 559.179,Z 218.833,A -85,B 0,C 180,E1 -3021.19,E2 -3021.19} C_VEL
LIN {X 0,Y 559.139,Z 218.84,A -85,B 0,C 180,E1 -3023.788,E2 -3023.788} C_VEL
LIN {X 0,Y 559.162,Z 218.835,A -85,B 0,C 180,E1 -3026.424,E2 -3026.424} C_VEL
LIN {X 0,Y 559.158,Z 218.837,A -85,B 0,C 180,E1 -3028.98,E2 -3028.98} C_VEL
LIN {X 0,Y 559.168,Z 218.835,A -85,B 0,C 180,E1 -3031.618,E2 -3031.618} C_VEL
LIN {X 0,Y 559.199,Z 218.831,A -85,B 0,C 180,E1 -3033.903,E2 -3033.903} C_VEL
LIN {X 0,Y 559.156,Z 218.837,A -85,B 0,C 180,E1 -3036.566,E2 -3036.566} C_VEL
LIN {X 0,Y 559.185,Z 218.834,A -85,B 0,C 180,E1 -3039.395,E2 -3039.395} C_VEL
LIN {X 0,Y 559.147,Z 218.838,A -85,B 0,C 180,E1 -3041.685,E2 -3041.685} C_VEL
LIN {X 0,Y 559.168,Z 218.834,A -85,B 0,C 180,E1 -3043.947,E2 -3043.947} C_VEL
LIN {X 0,Y 559.172,Z 218.834,A -85,B 0,C 180,E1 -3046.183,E2 -3046.183} C_VEL
LIN {X 0,Y 559.203,Z 218.831,A -85,B 0,C 180,E1 -3048.603,E2 -3048.603} C_VEL
LIN {X 0,Y 559.186,Z 218.832,A -85,B 0,C 180,E1 -3051.325,E2 -3051.325} C_VEL
LIN {X 0,Y 559.231,Z 218.828,A -85,B 0,C 180,E1 -3054.229,E2 -3054.229} C_VEL
LIN {X 0,Y 559.249,Z 218.824,A -85,B 0,C 180,E1 -3057.838,E2 -3057.838} C_VEL
LIN {X 0,Y 559.273,Z 218.821,A -85,B 0,C 180,E1 -3060.719,E2 -3060.719} C_VEL
LIN {X 0,Y 559.237,Z 218.826,A -85,B 0,C 180,E1 -3062.88,E2 -3062.88} C_VEL
LIN {X 0,Y 559.224,Z 218.829,A -85,B 0,C 180,E1 -3065.769,E2 -3065.769} C_VEL
LIN {X 0,Y 559.199,Z 218.833,A -85,B 0,C 180,E1 -3068.673,E2 -3068.673} C_VEL
LIN {X 0,Y 559.118,Z 218.843,A -85,B 0,C 180,E1 -3071.601,E2 -3071.601} C_VEL
LIN {X 0,Y 558.978,Z 219.098,A -85,B 0,C 180,E1 -3073.079,E2 -3073.079} C_VEL
LIN {X 0,Y 558.975,Z 221.697,A -85,B 0,C 180,E1 -3075.308,E2 -3075.308} C_VEL
LIN {X 0,Y 558.945,Z 224.311,A -85,B 0,C 180,E1 -3077.562,E2 -3077.562} C_VEL
LIN {X 0,Y 558.934,Z 226.914,A -85,B 0,C 180,E1 -3079.845,E2 -3079.845} C_VEL
LIN {X 0,Y 558.86,Z 230.406,A -85,B 0,C 180,E1 -3082.943,E2 -3082.943} C_VEL
LIN {X 0,Y 558.813,Z 233.048,A -85,B 0,C 180,E1 -3085.314,E2 -3085.314} C_VEL
LIN {X 0,Y 558.773,Z 235.833,A -85,B 0,C 180,E1 -3087.732,E2 -3087.732} C_VEL
LIN {X 0,Y 558.748,Z 238.855,A -85,B 0,C 180,E1 -3090.465,E2 -3090.465} C_VEL
LIN {X 0,Y 558.058,Z 239.595,A -85,B 0,C 180,E1 -3091.062,E2 -3091.062} C_VEL
LIN {X 0,Y 555.162,Z 240.948,A -85,B 0,C 180,E1 -3092.029,E2 -3092.029} C_VEL
LIN {X 0,Y 552.738,Z 242.051,A -85,B 0,C 180,E1 -3092.807,E2 -3092.807} C_VEL
LIN {X 0,Y 551.719,Z 242.842,A -85,B 0,C 180,E1 -3093.408,E2 -3093.408} C_VEL
LIN {X 0,Y 551.648,Z 243.092,A -85,B 0,C 180,E1 -3093.612,E2 -3093.612} C_VEL
LIN {X 0,Y 551.677,Z 243.681,A -85,B 0,C 180,E1 -3094.102,E2 -3094.102} C_VEL
LIN {X 0,Y 553.023,Z 252.878,A -85,B 0,C 180,E1 -3094.353,E2 -3094.353} C_VEL
LIN {X 0,Y 552.868,Z 265.649,A -85,B 0,C 180,E1 -3094.779,E2 -3094.779} C_VEL
LIN {X 0,Y 552.65,Z 278.712,A -85,B 0,C 180,E1 -3095.386,E2 -3095.386} C_VEL
LIN {X 0,Y 552.438,Z 289.534,A -85,B 0,C 180,E1 -3096.04,E2 -3096.04} C_VEL
LIN {X 0,Y 552.292,Z 300.106,A -85,B 0,C 180,E1 -3096.844,E2 -3096.844} C_VEL
LIN {X 0,Y 552.139,Z 310.549,A -85,B 0,C 180,E1 -3097.831,E2 -3097.831} C_VEL
LIN {X 0,Y 551.988,Z 319.031,A -85,B 0,C 180,E1 -3098.819,E2 -3098.819} C_VEL
LIN {X 0,Y 551.873,Z 326.286,A -85,B 0,C 180,E1 -3099.857,E2 -3099.857} C_VEL
LIN {X 0,Y 551.797,Z 332.183,A -85,B 0,C 180,E1 -3100.893,E2 -3100.893} C_VEL
LIN {X 0,Y 551.777,Z 336.914,A -85,B 0,C 180,E1 -3101.921,E2 -3101.921} C_VEL
LIN {X 0,Y 551.715,Z 340.654,A -85,B 0,C 180,E1 -3102.95,E2 -3102.95} C_VEL
LIN {X 0,Y 551.707,Z 343.43,A -85,B 0,C 180,E1 -3103.965,E2 -3103.965} C_VEL
LIN {X 0,Y 551.687,Z 344.542,A -85,B 0,C 180,E1 -3104.49,E2 -3104.49} C_VEL
LIN {X 0,Y 551.688,Z 346.115,A -85,B 0,C 180,E1 -3105.522,E2 -3105.522} C_VEL
LIN {X 0,Y 551.655,Z 346.902,A -85,B 0,C 180,E1 -3106.564,E2 -3106.564} C_VEL
LIN {X 0,Y 551.642,Z 346.869,A -85,B 0,C 180,E1 -3107.637,E2 -3107.637} C_VEL
LIN {X 0,Y 551.658,Z 345.936,A -85,B 0,C 180,E1 -3108.73,E2 -3108.73} C_VEL
LIN {X 0,Y 551.662,Z 344.046,A -85,B 0,C 180,E1 -3109.849,E2 -3109.849} C_VEL
LIN {X 0,Y 551.729,Z 341.117,A -85,B 0,C 180,E1 -3110.986,E2 -3110.986} C_VEL
LIN {X 0,Y 551.752,Z 336.322,A -85,B 0,C 180,E1 -3112.31,E2 -3112.31} C_VEL
LIN {X 0,Y 551.837,Z 330.287,A -85,B 0,C 180,E1 -3113.55,E2 -3113.55} C_VEL
LIN {X 0,Y 551.888,Z 323.971,A -85,B 0,C 180,E1 -3114.585,E2 -3114.585} C_VEL
LIN {X 0,Y 552.057,Z 315.732,A -85,B 0,C 180,E1 -3115.68,E2 -3115.68} C_VEL
LIN {X 0,Y 552.226,Z 306.017,A -85,B 0,C 180,E1 -3116.713,E2 -3116.713} C_VEL
LIN {X 0,Y 552.375,Z 295.669,A -85,B 0,C 180,E1 -3117.603,E2 -3117.603} C_VEL
LIN {X 0,Y 552.572,Z 284.463,A -85,B 0,C 180,E1 -3118.375,E2 -3118.375} C_VEL
LIN {X 0,Y 552.736,Z 272.699,A -85,B 0,C 180,E1 -3119.006,E2 -3119.006} C_VEL
LIN {X 0,Y 552.968,Z 259.565,A -85,B 0,C 180,E1 -3119.534,E2 -3119.534} C_VEL
LIN {X 0,Y 552.864,Z 250.72,A -85,B 0,C 180,E1 -3119.796,E2 -3119.796} C_VEL
LIN {X 0,Y 551.693,Z 243.664,A -85,B 0,C 180,E1 -3120.001,E2 -3120.001} C_VEL
LIN {X 0,Y 551.719,Z 239.964,A -85,B 0,C 180,E1 -3123.081,E2 -3123.081} C_VEL
LIN {X 0,Y 551.728,Z 236.66,A -85,B 0,C 180,E1 -3125.945,E2 -3125.945} C_VEL
LIN {X 0,Y 551.754,Z 233.906,A -85,B 0,C 180,E1 -3128.405,E2 -3128.405} C_VEL
LIN {X 0,Y 551.777,Z 230.39,A -85,B 0,C 180,E1 -3131.433,E2 -3131.433} C_VEL
LIN {X 0,Y 551.798,Z 227.729,A -85,B 0,C 180,E1 -3133.728,E2 -3133.728} C_VEL
LIN {X 0,Y 551.86,Z 225.142,A -85,B 0,C 180,E1 -3135.998,E2 -3135.998} C_VEL
LIN {X 0,Y 551.92,Z 221.653,A -85,B 0,C 180,E1 -3138.989,E2 -3138.989} C_VEL
LIN {X 0,Y 551.864,Z 219.937,A -85,B 0,C 180,E1 -3140.471,E2 -3140.471} C_VEL
LIN {X 0,Y 552.174,Z 219.705,A -85,B 0,C 180,E1 -3143.091,E2 -3143.091} C_VEL
LIN {X 0,Y 552.222,Z 219.701,A -85,B 0,C 180,E1 -3144.889,E2 -3144.889} C_VEL
LIN {X 0,Y 552.21,Z 219.701,A -85,B 0,C 180,E1 -3147.812,E2 -3147.812} C_VEL
LIN {X 0,Y 552.236,Z 219.7,A -85,B 0,C 180,E1 -3150.73,E2 -3150.73} C_VEL
LIN {X 0,Y 552.194,Z 219.704,A -85,B 0,C 180,E1 -3152.919,E2 -3152.919} C_VEL
LIN {X 0,Y 552.188,Z 219.703,A -85,B 0,C 180,E1 -3155.844,E2 -3155.844} C_VEL
LIN {X 0,Y 552.156,Z 219.708,A -85,B 0,C 180,E1 -3158.786,E2 -3158.786} C_VEL
LIN {X 0,Y 552.149,Z 219.708,A -85,B 0,C 180,E1 -3161.751,E2 -3161.751} C_VEL
LIN {X 0,Y 552.121,Z 219.713,A -85,B 0,C 180,E1 -3164.749,E2 -3164.749} C_VEL
LIN {X 0,Y 552.104,Z 219.713,A -85,B 0,C 180,E1 -3167.789,E2 -3167.789} C_VEL
LIN {X 0,Y 552.121,Z 219.712,A -85,B 0,C 180,E1 -3170.102,E2 -3170.102} C_VEL
LIN {X 0,Y 552.102,Z 219.715,A -85,B 0,C 180,E1 -3172.451,E2 -3172.451} C_VEL
LIN {X 0,Y 552.149,Z 219.709,A -85,B 0,C 180,E1 -3175.353,E2 -3175.353} C_VEL
LIN {X 0,Y 552.115,Z 219.715,A -85,B 0,C 180,E1 -3178.098,E2 -3178.098} C_VEL
LIN {X 0,Y 552.095,Z 219.717,A -85,B 0,C 180,E1 -3180.61,E2 -3180.61} C_VEL
LIN {X 0,Y 552.117,Z 219.712,A -85,B 0,C 180,E1 -3183.186,E2 -3183.186} C_VEL
LIN {X 0,Y 552.1,Z 219.713,A -85,B 0,C 180,E1 -3185.843,E2 -3185.843} C_VEL
LIN {X 0,Y 552.116,Z 219.713,A -85,B 0,C 180,E1 -3189.063,E2 -3189.063} C_VEL
LIN {X 0,Y 552.16,Z 219.707,A -85,B 0,C 180,E1 -3191.443,E2 -3191.443} C_VEL
LIN {X 0,Y 552.087,Z 219.717,A -85,B 0,C 180,E1 -3194.533,E2 -3194.533} C_VEL
LIN {X 0,Y 552.122,Z 219.711,A -85,B 0,C 180,E1 -3197.586,E2 -3197.586} C_VEL
LIN {X 0,Y 552.128,Z 219.712,A -85,B 0,C 180,E1 -3200.475,E2 -3200.475} C_VEL
LIN {X 0,Y 552.107,Z 219.714,A -85,B 0,C 180,E1 -3203.317,E2 -3203.317} C_VEL
LIN {X 0,Y 552.131,Z 219.71,A -85,B 0,C 180,E1 -3205.941,E2 -3205.941} C_VEL
LIN {X 0,Y 552.113,Z 219.713,A -85,B 0,C 180,E1 -3208.542,E2 -3208.542} C_VEL
LIN {X 0,Y 552.122,Z 219.714,A -85,B 0,C 180,E1 -3211.439,E2 -3211.439} C_VEL
LIN {X 0,Y 552.126,Z 219.711,A -85,B 0,C 180,E1 -3214.357,E2 -3214.357} C_VEL
LIN {X 0,Y 552.107,Z 219.713,A -85,B 0,C 180,E1 -3216.76,E2 -3216.76} C_VEL
LIN {X 0,Y 552.118,Z 219.711,A -85,B 0,C 180,E1 -3219.121,E2 -3219.121} C_VEL
LIN {X 0,Y 552.129,Z 219.71,A -85,B 0,C 180,E1 -3221.446,E2 -3221.446} C_VEL
LIN {X 0,Y 552.119,Z 219.712,A -85,B 0,C 180,E1 -3223.739,E2 -3223.739} C_VEL
LIN {X 0,Y 552.135,Z 219.711,A -85,B 0,C 180,E1 -3226.006,E2 -3226.006} C_VEL
LIN {X 0,Y 552.163,Z 219.707,A -85,B 0,C 180,E1 -3228.995,E2 -3228.995} C_VEL
LIN {X 0,Y 552.146,Z 219.709,A -85,B 0,C 180,E1 -3231.953,E2 -3231.953} C_VEL
LIN {X 0,Y 552.229,Z 219.698,A -85,B 0,C 180,E1 -3234.89,E2 -3234.89} C_VEL
LIN {X 0,Y 552.219,Z 219.701,A -85,B 0,C 180,E1 -3237.813,E2 -3237.813} C_VEL
LIN {X 0,Y 552.24,Z 219.696,A -85,B 0,C 180,E1 -3240.73,E2 -3240.73} C_VEL
LIN {X 0,Y 552.206,Z 219.701,A -85,B 0,C 180,E1 -3242.919,E2 -3242.919} C_VEL
LIN {X 0,Y 552.195,Z 219.705,A -85,B 0,C 180,E1 -3245.845,E2 -3245.845} C_VEL
LIN {X 0,Y 552.145,Z 219.708,A -85,B 0,C 180,E1 -3248.787,E2 -3248.787} C_VEL
LIN {X 0,Y 552.167,Z 219.708,A -85,B 0,C 180,E1 -3251.751,E2 -3251.751} C_VEL
LIN {X 0,Y 552.141,Z 219.709,A -85,B 0,C 180,E1 -3254.749,E2 -3254.749} C_VEL
LIN {X 0,Y 552.117,Z 219.715,A -85,B 0,C 180,E1 -3257.789,E2 -3257.789} C_VEL
LIN {X 0,Y 552.131,Z 219.712,A -85,B 0,C 180,E1 -3260.102,E2 -3260.102} C_VEL
LIN {X 0,Y 552.097,Z 219.716,A -85,B 0,C 180,E1 -3262.452,E2 -3262.452} C_VEL
LIN {X 0,Y 552.114,Z 219.712,A -85,B 0,C 180,E1 -3265.646,E2 -3265.646} C_VEL
LIN {X 0,Y 552.125,Z 219.71,A -85,B 0,C 180,E1 -3268.098,E2 -3268.098} C_VEL
LIN {X 0,Y 552.103,Z 219.713,A -85,B 0,C 180,E1 -3270.61,E2 -3270.61} C_VEL
LIN {X 0,Y 552.113,Z 219.714,A -85,B 0,C 180,E1 -3273.187,E2 -3273.187} C_VEL
LIN {X 0,Y 552.091,Z 219.717,A -85,B 0,C 180,E1 -3275.844,E2 -3275.844} C_VEL
LIN {X 0,Y 552.123,Z 219.712,A -85,B 0,C 180,E1 -3278.589,E2 -3278.589} C_VEL
LIN {X 0,Y 552.126,Z 219.712,A -85,B 0,C 180,E1 -3281.446,E2 -3281.446} C_VEL
LIN {X 0,Y 552.099,Z 219.714,A -85,B 0,C 180,E1 -3284.532,E2 -3284.532} C_VEL
LIN {X 0,Y 552.136,Z 219.712,A -85,B 0,C 180,E1 -3287.585,E2 -3287.585} C_VEL
LIN {X 0,Y 552.138,Z 219.712,A -85,B 0,C 180,E1 -3290.473,E2 -3290.473} C_VEL
LIN {X 0,Y 552.127,Z 219.806,A -85,B 0,C 180,E1 -3292.511,E2 -3292.511} C_VEL
LIN {X 0,Y 552.916,Z 225.235,A -85,B 0,C 180,E1 -3294.439,E2 -3294.439} C_VEL
LIN {X 0,Y 552.853,Z 232.507,A -85,B 0,C 180,E1 -3296.864,E2 -3296.864} C_VEL
LIN {X 0,Y 552.661,Z 241.794,A -85,B 0,C 180,E1 -3299.853,E2 -3299.853} C_VEL
LIN {X 0,Y 552.488,Z 251.041,A -85,B 0,C 180,E1 -3302.745,E2 -3302.745} C_VEL
LIN {X 0,Y 552.353,Z 260.309,A -85,B 0,C 180,E1 -3305.573,E2 -3305.573} C_VEL
LIN {X 0,Y 552.214,Z 269.576,A -85,B 0,C 180,E1 -3308.341,E2 -3308.341} C_VEL
LIN {X 0,Y 552.087,Z 278.843,A -85,B 0,C 180,E1 -3311.058,E2 -3311.058} C_VEL
LIN {X 0,Y 551.994,Z 289.434,A -85,B 0,C 180,E1 -3314.113,E2 -3314.113} C_VEL
LIN {X 0,Y 551.888,Z 299.529,A -85,B 0,C 180,E1 -3316.983,E2 -3316.983} C_VEL
LIN {X 0,Y 553.101,Z 308.509,A -85,B 0,C 180,E1 -3317.198,E2 -3317.198} C_VEL
LIN {X 0,Y 552.929,Z 321.168,A -85,B 0,C 180,E1 -3317.567,E2 -3317.567} C_VEL
LIN {X 0,Y 552.743,Z 333.478,A -85,B 0,C 180,E1 -3318.076,E2 -3318.076} C_VEL
LIN {X 0,Y 552.578,Z 345.229,A -85,B 0,C 180,E1 -3318.717,E2 -3318.717} C_VEL
LIN {X 0,Y 552.441,Z 355.923,A -85,B 0,C 180,E1 -3319.462,E2 -3319.462} C_VEL
LIN {X 0,Y 552.234,Z 365.597,A -85,B 0,C 180,E1 -3320.292,E2 -3320.292} C_VEL
LIN {X 0,Y 552.077,Z 374.41,A -85,B 0,C 180,E1 -3321.213,E2 -3321.213} C_VEL
LIN {X 0,Y 551.951,Z 382.998,A -85,B 0,C 180,E1 -3322.316,E2 -3322.316} C_VEL
LIN {X 0,Y 551.825,Z 389.865,A -85,B 0,C 180,E1 -3323.418,E2 -3323.418} C_VEL
LIN {X 0,Y 551.804,Z 395.364,A -85,B 0,C 180,E1 -3324.518,E2 -3324.518} C_VEL
LIN {X 0,Y 551.764,Z 399.676,A -85,B 0,C 180,E1 -3325.617,E2 -3325.617} C_VEL
LIN {X 0,Y 551.751,Z 401.956,A -85,B 0,C 180,E1 -3326.348,E2 -3326.348} C_VEL
LIN {X 0,Y 551.724,Z 403.807,A -85,B 0,C 180,E1 -3327.079,E2 -3327.079} C_VEL
LIN {X 0,Y 551.657,Z 405.198,A -85,B 0,C 180,E1 -3327.809,E2 -3327.809} C_VEL
LIN {X 0,Y 551.641,Z 406.784,A -85,B 0,C 180,E1 -3329.27,E2 -3329.27} C_VEL
LIN {X 0,Y 551.64,Z 407,A -85,B 0,C 180,E1 -3330,E2 -3330} C_VEL
LIN {X 0,Y 551.645,Z 406.186,A -85,B 0,C 180,E1 -3331.46,E2 -3331.46} C_VEL
LIN {X 0,Y 551.657,Z 405.201,A -85,B 0,C 180,E1 -3332.19,E2 -3332.19} C_VEL
LIN {X 0,Y 551.724,Z 403.811,A -85,B 0,C 180,E1 -3332.92,E2 -3332.92} C_VEL
LIN {X 0,Y 551.764,Z 400.897,A -85,B 0,C 180,E1 -3334.017,E2 -3334.017} C_VEL
LIN {X 0,Y 551.724,Z 396.951,A -85,B 0,C 180,E1 -3335.115,E2 -3335.115} C_VEL
LIN {X 0,Y 551.823,Z 391.207,A -85,B 0,C 180,E1 -3336.338,E2 -3336.338} C_VEL
LIN {X 0,Y 551.927,Z 384.24,A -85,B 0,C 180,E1 -3337.499,E2 -3337.499} C_VEL
LIN {X 0,Y 552.082,Z 375.994,A -85,B 0,C 180,E1 -3338.602,E2 -3338.602} C_VEL
LIN {X 0,Y 552.201,Z 367.543,A -85,B 0,C 180,E1 -3339.523,E2 -3339.523} C_VEL
LIN {X 0,Y 552.404,Z 357.102,A -85,B 0,C 180,E1 -3340.445,E2 -3340.445} C_VEL
LIN {X 0,Y 552.556,Z 346.375,A -85,B 0,C 180,E1 -3341.209,E2 -3341.209} C_VEL
LIN {X 0,Y 552.704,Z 335.421,A -85,B 0,C 180,E1 -3341.831,E2 -3341.831} C_VEL
LIN {X 0,Y 552.898,Z 323.776,A -85,B 0,C 180,E1 -3342.339,E2 -3342.339} C_VEL
LIN {X 0,Y 553.068,Z 310.368,A -85,B 0,C 180,E1 -3342.755,E2 -3342.755} C_VEL
LIN {X 0,Y 552.894,Z 305.824,A -85,B 0,C 180,E1 -3342.864,E2 -3342.864} C_VEL
LIN {X 0,Y 551.888,Z 299.532,A -85,B 0,C 180,E1 -3343.017,E2 -3343.017} C_VEL
LIN {X 0,Y 551.994,Z 289.437,A -85,B 0,C 180,E1 -3345.886,E2 -3345.886} C_VEL
LIN {X 0,Y 552.085,Z 278.846,A -85,B 0,C 180,E1 -3348.942,E2 -3348.942} C_VEL
LIN {X 0,Y 552.254,Z 268.256,A -85,B 0,C 180,E1 -3352.049,E2 -3352.049} C_VEL
LIN {X 0,Y 552.367,Z 258.988,A -85,B 0,C 180,E1 -3354.826,E2 -3354.826} C_VEL
LIN {X 0,Y 552.525,Z 249.72,A -85,B 0,C 180,E1 -3357.663,E2 -3357.663} C_VEL
LIN {X 0,Y 552.67,Z 240.453,A -85,B 0,C 180,E1 -3360.574,E2 -3360.574} C_VEL
LIN {X 0,Y 552.898,Z 231.186,A -85,B 0,C 180,E1 -3363.568,E2 -3363.568} C_VEL
LIN {X 0,Y 552.886,Z 224.436,A -85,B 0,C 180,E1 -3365.783,E2 -3365.783} C_VEL
LIN {X 0,Y 552.112,Z 219.716,A -85,B 0,C 180,E1 -3367.546,E2 -3367.546} C_VEL
LIN {X 0,Y 552.11,Z 219.716,A -85,B 0,C 180,E1 -3370.48,E2 -3370.48} C_VEL
LIN {X 0,Y 552.12,Z 219.715,A -85,B 0,C 180,E1 -3373.484,E2 -3373.484} C_VEL
LIN {X 0,Y 552.107,Z 219.716,A -85,B 0,C 180,E1 -3376.575,E2 -3376.575} C_VEL
LIN {X 0,Y 552.143,Z 219.711,A -85,B 0,C 180,E1 -3379.521,E2 -3379.521} C_VEL
LIN {X 0,Y 552.095,Z 219.716,A -85,B 0,C 180,E1 -3382.335,E2 -3382.335} C_VEL
LIN {X 0,Y 552.085,Z 219.719,A -85,B 0,C 180,E1 -3385.05,E2 -3385.05} C_VEL
LIN {X 0,Y 552.115,Z 219.713,A -85,B 0,C 180,E1 -3387.68,E2 -3387.68} C_VEL
LIN {X 0,Y 552.112,Z 219.715,A -85,B 0,C 180,E1 -3390.234,E2 -3390.234} C_VEL
LIN {X 0,Y 552.146,Z 219.71,A -85,B 0,C 180,E1 -3392.997,E2 -3392.997} C_VEL
LIN {X 0,Y 552.113,Z 219.714,A -85,B 0,C 180,E1 -3395.16,E2 -3395.16} C_VEL
LIN {X 0,Y 552.096,Z 219.716,A -85,B 0,C 180,E1 -3397.548,E2 -3397.548} C_VEL
LIN {X 0,Y 552.149,Z 219.709,A -85,B 0,C 180,E1 -3400.372,E2 -3400.372} C_VEL
LIN {X 0,Y 552.155,Z 219.708,A -85,B 0,C 180,E1 -3402.976,E2 -3402.976} C_VEL
LIN {X 0,Y 552.135,Z 219.711,A -85,B 0,C 180,E1 -3406.003,E2 -3406.003} C_VEL
LIN {X 0,Y 552.159,Z 219.708,A -85,B 0,C 180,E1 -3408.992,E2 -3408.992} C_VEL
LIN {X 0,Y 552.16,Z 219.709,A -85,B 0,C 180,E1 -3411.95,E2 -3411.95} C_VEL
LIN {X 0,Y 552.228,Z 219.7,A -85,B 0,C 180,E1 -3414.888,E2 -3414.888} C_VEL
LIN {X 0,Y 552.22,Z 219.699,A -85,B 0,C 180,E1 -3417.811,E2 -3417.811} C_VEL
LIN {X 0,Y 552.242,Z 219.697,A -85,B 0,C 180,E1 -3420.728,E2 -3420.728} C_VEL
LIN {X 0,Y 552.204,Z 219.702,A -85,B 0,C 180,E1 -3422.917,E2 -3422.917} C_VEL
LIN {X 0,Y 552.195,Z 219.704,A -85,B 0,C 180,E1 -3425.843,E2 -3425.843} C_VEL
LIN {X 0,Y 552.167,Z 219.708,A -85,B 0,C 180,E1 -3428.784,E2 -3428.784} C_VEL
LIN {X 0,Y 552.057,Z 219.724,A -85,B 0,C 180,E1 -3431.751,E2 -3431.751} C_VEL
LIN {X 0,Y 551.911,Z 220.027,A -85,B 0,C 180,E1 -3433.249,E2 -3433.249} C_VEL
LIN {X 0,Y 551.911,Z 222.628,A -85,B 0,C 180,E1 -3435.509,E2 -3435.509} C_VEL
LIN {X 0,Y 551.888,Z 225.259,A -85,B 0,C 180,E1 -3437.794,E2 -3437.794} C_VEL
LIN {X 0,Y 551.857,Z 227.893,A -85,B 0,C 180,E1 -3440.11,E2 -3440.11} C_VEL
LIN {X 0,Y 551.809,Z 231.393,A -85,B 0,C 180,E1 -3443.253,E2 -3443.253} C_VEL
LIN {X 0,Y 551.74,Z 234.115,A -85,B 0,C 180,E1 -3445.662,E2 -3445.662} C_VEL
LIN {X 0,Y 551.725,Z 236.922,A -85,B 0,C 180,E1 -3448.118,E2 -3448.118} C_VEL
LIN {X 0,Y 551.671,Z 239.687,A -85,B 0,C 180,E1 -3450.634,E2 -3450.634} C_VEL
LIN {X 0,Y 551.648,Z 243.092,A -85,B 0,C 180,E1 -3453.612,E2 -3453.612} C_VEL
LIN {X 0,Y 551.578,Z 244.277,A -85,B 0,C 180,E1 -3453.867,E2 -3453.867} C_VEL
LIN {X 0,Y 551.326,Z 247.054,A -85,B 0,C 180,E1 -3454.088,E2 -3454.088} C_VEL
LIN {X 0,Y 550.725,Z 251.904,A -85,B 0,C 180,E1 -3454.274,E2 -3454.274} C_VEL
LIN {X 0,Y 548.948,Z 260.229,A -85,B 0,C 180,E1 -3454.486,E2 -3454.486} C_VEL
LIN {X 0,Y 546.265,Z 268.945,A -85,B 0,C 180,E1 -3454.756,E2 -3454.756} C_VEL
LIN {X 0,Y 545.851,Z 271.815,A -85,B 0,C 180,E1 -3454.882,E2 -3454.882} C_VEL
LIN {X 0,Y 545.618,Z 283.431,A -85,B 0,C 180,E1 -3455.501,E2 -3455.501} C_VEL
LIN {X 0,Y 545.382,Z 294.698,A -85,B 0,C 180,E1 -3456.268,E2 -3456.268} C_VEL
LIN {X 0,Y 545.182,Z 305.404,A -85,B 0,C 180,E1 -3457.192,E2 -3457.192} C_VEL
LIN {X 0,Y 545.006,Z 315.245,A -85,B 0,C 180,E1 -3458.239,E2 -3458.239} C_VEL
LIN {X 0,Y 544.862,Z 323.219,A -85,B 0,C 180,E1 -3459.294,E2 -3459.294} C_VEL
LIN {X 0,Y 544.723,Z 330.153,A -85,B 0,C 180,E1 -3460.429,E2 -3460.429} C_VEL
LIN {X 0,Y 544.705,Z 335.635,A -85,B 0,C 180,E1 -3461.554,E2 -3461.554} C_VEL
LIN {X 0,Y 544.655,Z 339.832,A -85,B 0,C 180,E1 -3462.651,E2 -3462.651} C_VEL
LIN {X 0,Y 544.616,Z 342.952,A -85,B 0,C 180,E1 -3463.727,E2 -3463.727} C_VEL
LIN {X 0,Y 544.573,Z 345.786,A -85,B 0,C 180,E1 -3465.216,E2 -3465.216} C_VEL
LIN {X 0,Y 544.561,Z 346.768,A -85,B 0,C 180,E1 -3466.277,E2 -3466.277} C_VEL
LIN {X 0,Y 544.532,Z 346.938,A -85,B 0,C 180,E1 -3467.361,E2 -3467.361} C_VEL
LIN {X 0,Y 544.554,Z 345.834,A -85,B 0,C 180,E1 -3468.838,E2 -3468.838} C_VEL
LIN {X 0,Y 544.599,Z 343.103,A -85,B 0,C 180,E1 -3470.299,E2 -3470.299} C_VEL
LIN {X 0,Y 544.652,Z 338.85,A -85,B 0,C 180,E1 -3471.73,E2 -3471.73} C_VEL
LIN {X 0,Y 544.699,Z 333.913,A -85,B 0,C 180,E1 -3472.922,E2 -3472.922} C_VEL
LIN {X 0,Y 544.807,Z 326.977,A -85,B 0,C 180,E1 -3474.211,E2 -3474.211} C_VEL
LIN {X 0,Y 544.938,Z 318.646,A -85,B 0,C 180,E1 -3475.427,E2 -3475.427} C_VEL
LIN {X 0,Y 545.11,Z 309.49,A -85,B 0,C 180,E1 -3476.49,E2 -3476.49} C_VEL
LIN {X 0,Y 545.307,Z 299.325,A -85,B 0,C 180,E1 -3477.448,E2 -3477.448} C_VEL
LIN {X 0,Y 545.513,Z 288.866,A -85,B 0,C 180,E1 -3478.24,E2 -3478.24} C_VEL
LIN {X 0,Y 545.735,Z 277.187,A -85,B 0,C 180,E1 -3478.941,E2 -3478.941} C_VEL
LIN {X 0,Y 545.986,Z 265.193,A -85,B 0,C 180,E1 -3479.493,E2 -3479.493} C_VEL
LIN {X 0,Y 546.064,Z 252.367,A -85,B 0,C 180,E1 -3479.919,E2 -3479.919} C_VEL
LIN {X 0,Y 544.587,Z 243.927,A -85,B 0,C 180,E1 -3480.156,E2 -3480.156} C_VEL
LIN {X 0,Y 544.637,Z 240.392,A -85,B 0,C 180,E1 -3483.152,E2 -3483.152} C_VEL
LIN {X 0,Y 544.653,Z 237.584,A -85,B 0,C 180,E1 -3485.612,E2 -3485.612} C_VEL
LIN {X 0,Y 544.668,Z 234.602,A -85,B 0,C 180,E1 -3488.279,E2 -3488.279} C_VEL
LIN {X 0,Y 544.701,Z 231.291,A -85,B 0,C 180,E1 -3491.183,E2 -3491.183} C_VEL
LIN {X 0,Y 544.739,Z 228.593,A -85,B 0,C 180,E1 -3493.511,E2 -3493.511} C_VEL
LIN {X 0,Y 544.783,Z 225.95,A -85,B 0,C 180,E1 -3495.812,E2 -3495.812} C_VEL
LIN {X 0,Y 544.878,Z 222.46,A -85,B 0,C 180,E1 -3498.845,E2 -3498.845} C_VEL
LIN {X 0,Y 544.791,Z 220.746,A -85,B 0,C 180,E1 -3500.346,E2 -3500.346} C_VEL
LIN {X 0,Y 545.142,Z 220.581,A -85,B 0,C 180,E1 -3503.05,E2 -3503.05} C_VEL
LIN {X 0,Y 545.196,Z 220.576,A -85,B 0,C 180,E1 -3504.823,E2 -3504.823} C_VEL
LIN {X 0,Y 545.181,Z 220.576,A -85,B 0,C 180,E1 -3507.784,E2 -3507.784} C_VEL
LIN {X 0,Y 545.205,Z 220.576,A -85,B 0,C 180,E1 -3510.739,E2 -3510.739} C_VEL
LIN {X 0,Y 545.16,Z 220.581,A -85,B 0,C 180,E1 -3512.956,E2 -3512.956} C_VEL
LIN {X 0,Y 545.159,Z 220.578,A -85,B 0,C 180,E1 -3515.92,E2 -3515.92} C_VEL
LIN {X 0,Y 545.113,Z 220.587,A -85,B 0,C 180,E1 -3518.901,E2 -3518.901} C_VEL
LIN {X 0,Y 545.121,Z 220.583,A -85,B 0,C 180,E1 -3521.905,E2 -3521.905} C_VEL
LIN {X 0,Y 545.071,Z 220.593,A -85,B 0,C 180,E1 -3524.944,E2 -3524.944} C_VEL
LIN {X 0,Y 545.071,Z 220.589,A -85,B 0,C 180,E1 -3528.026,E2 -3528.026} C_VEL
LIN {X 0,Y 545.086,Z 220.588,A -85,B 0,C 180,E1 -3530.373,E2 -3530.373} C_VEL
LIN {X 0,Y 545.1,Z 220.586,A -85,B 0,C 180,E1 -3533.559,E2 -3533.559} C_VEL
LIN {X 0,Y 545.078,Z 220.589,A -85,B 0,C 180,E1 -3536.001,E2 -3536.001} C_VEL
LIN {X 0,Y 545.078,Z 220.589,A -85,B 0,C 180,E1 -3538.75,E2 -3538.75} C_VEL
LIN {X 0,Y 545.066,Z 220.592,A -85,B 0,C 180,E1 -3541.684,E2 -3541.684} C_VEL
LIN {X 0,Y 545.073,Z 220.59,A -85,B 0,C 180,E1 -3544.564,E2 -3544.564} C_VEL
LIN {X 0,Y 545.028,Z 220.596,A -85,B 0,C 180,E1 -3547.305,E2 -3547.305} C_VEL
LIN {X 0,Y 545.084,Z 220.59,A -85,B 0,C 180,E1 -3550.141,E2 -3550.141} C_VEL
LIN {X 0,Y 545.057,Z 220.592,A -85,B 0,C 180,E1 -3552.699,E2 -3552.699} C_VEL
LIN {X 0,Y 545.054,Z 220.591,A -85,B 0,C 180,E1 -3555.168,E2 -3555.168} C_VEL
LIN {X 0,Y 545.074,Z 220.589,A -85,B 0,C 180,E1 -3557.899,E2 -3557.899} C_VEL
LIN {X 0,Y 545.099,Z 220.589,A -85,B 0,C 180,E1 -3560.677,E2 -3560.677} C_VEL
LIN {X 0,Y 545.047,Z 220.592,A -85,B 0,C 180,E1 -3563.622,E2 -3563.622} C_VEL
LIN {X 0,Y 545.07,Z 220.591,A -85,B 0,C 180,E1 -3566.331,E2 -3566.331} C_VEL
LIN {X 0,Y 545.065,Z 220.593,A -85,B 0,C 180,E1 -3568.954,E2 -3568.954} C_VEL
LIN {X 0,Y 545.1,Z 220.588,A -85,B 0,C 180,E1 -3571.509,E2 -3571.509} C_VEL
LIN {X 0,Y 545.091,Z 220.587,A -85,B 0,C 180,E1 -3574.493,E2 -3574.493} C_VEL
LIN {X 0,Y 545.042,Z 220.595,A -85,B 0,C 180,E1 -3577.244,E2 -3577.244} C_VEL
LIN {X 0,Y 545.118,Z 220.584,A -85,B 0,C 180,E1 -3580.416,E2 -3580.416} C_VEL
LIN {X 0,Y 545.075,Z 220.591,A -85,B 0,C 180,E1 -3583.523,E2 -3583.523} C_VEL
LIN {X 0,Y 545.094,Z 220.589,A -85,B 0,C 180,E1 -3585.821,E2 -3585.821} C_VEL
LIN {X 0,Y 545.119,Z 220.583,A -85,B 0,C 180,E1 -3588.851,E2 -3588.851} C_VEL
LIN {X 0,Y 545.095,Z 220.589,A -85,B 0,C 180,E1 -3591.848,E2 -3591.848} C_VEL
LIN {X 0,Y 545.205,Z 220.573,A -85,B 0,C 180,E1 -3594.824,E2 -3594.824} C_VEL
LIN {X 0,Y 545.191,Z 220.577,A -85,B 0,C 180,E1 -3597.785,E2 -3597.785} C_VEL
LIN {X 0,Y 545.211,Z 220.572,A -85,B 0,C 180,E1 -3600.74,E2 -3600.74} C_VEL
LIN {X 0,Y 545.173,Z 220.577,A -85,B 0,C 180,E1 -3602.957,E2 -3602.957} C_VEL
LIN {X 0,Y 545.166,Z 220.581,A -85,B 0,C 180,E1 -3605.921,E2 -3605.921} C_VEL
LIN {X 0,Y 545.105,Z 220.585,A -85,B 0,C 180,E1 -3608.901,E2 -3608.901} C_VEL
LIN {X 0,Y 545.139,Z 220.584,A -85,B 0,C 180,E1 -3611.905,E2 -3611.905} C_VEL
LIN {X 0,Y 545.09,Z 220.587,A -85,B 0,C 180,E1 -3614.944,E2 -3614.944} C_VEL
LIN {X 0,Y 545.085,Z 220.589,A -85,B 0,C 180,E1 -3618.027,E2 -3618.027} C_VEL
LIN {X 0,Y 545.097,Z 220.588,A -85,B 0,C 180,E1 -3620.373,E2 -3620.373} C_VEL
LIN {X 0,Y 545.081,Z 220.59,A -85,B 0,C 180,E1 -3623.56,E2 -3623.56} C_VEL
LIN {X 0,Y 545.074,Z 220.591,A -85,B 0,C 180,E1 -3626.002,E2 -3626.002} C_VEL
LIN {X 0,Y 545.094,Z 220.589,A -85,B 0,C 180,E1 -3628.749,E2 -3628.749} C_VEL
LIN {X 0,Y 545.06,Z 220.592,A -85,B 0,C 180,E1 -3631.915,E2 -3631.915} C_VEL
LIN {X 0,Y 545.065,Z 220.592,A -85,B 0,C 180,E1 -3634.565,E2 -3634.565} C_VEL
LIN {X 0,Y 545.042,Z 220.594,A -85,B 0,C 180,E1 -3637.304,E2 -3637.304} C_VEL
LIN {X 0,Y 545.071,Z 220.589,A -85,B 0,C 180,E1 -3640.143,E2 -3640.143} C_VEL
LIN {X 0,Y 545.084,Z 220.589,A -85,B 0,C 180,E1 -3643.107,E2 -3643.107} C_VEL
LIN {X 0,Y 545.055,Z 220.592,A -85,B 0,C 180,E1 -3646.227,E2 -3646.227} C_VEL
LIN {X 0,Y 545.087,Z 220.591,A -85,B 0,C 180,E1 -3648.886,E2 -3648.886} C_VEL
LIN {X 0,Y 545.088,Z 220.59,A -85,B 0,C 180,E1 -3650.819,E2 -3650.819} C_VEL
LIN {X 0,Y 545.057,Z 220.646,A -85,B 0,C 180,E1 -3652.232,E2 -3652.232} C_VEL
LIN {X 0,Y 545.976,Z 226.044,A -85,B 0,C 180,E1 -3654.191,E2 -3654.191} C_VEL
LIN {X 0,Y 545.888,Z 233.781,A -85,B 0,C 180,E1 -3656.809,E2 -3656.809} C_VEL
LIN {X 0,Y 545.667,Z 243.098,A -85,B 0,C 180,E1 -3659.847,E2 -3659.847} C_VEL
LIN {X 0,Y 545.506,Z 252.241,A -85,B 0,C 180,E1 -3662.744,E2 -3662.744} C_VEL
LIN {X 0,Y 545.343,Z 261.633,A -85,B 0,C 180,E1 -3665.644,E2 -3665.644} C_VEL
LIN {X 0,Y 545.174,Z 271.063,A -85,B 0,C 180,E1 -3668.493,E2 -3668.493} C_VEL
LIN {X 0,Y 545.031,Z 280.167,A -85,B 0,C 180,E1 -3671.194,E2 -3671.194} C_VEL
LIN {X 0,Y 544.922,Z 290.758,A -85,B 0,C 180,E1 -3674.285,E2 -3674.285} C_VEL
LIN {X 0,Y 544.804,Z 299.529,A -85,B 0,C 180,E1 -3676.81,E2 -3676.81} C_VEL
LIN {X 0,Y 546.181,Z 309.424,A -85,B 0,C 180,E1 -3677.057,E2 -3677.057} C_VEL
LIN {X 0,Y 545.975,Z 322.464,A -85,B 0,C 180,E1 -3677.454,E2 -3677.454} C_VEL
LIN {X 0,Y 545.783,Z 333.479,A -85,B 0,C 180,E1 -3677.921,E2 -3677.921} C_VEL
LIN {X 0,Y 545.585,Z 345.612,A -85,B 0,C 180,E1 -3678.595,E2 -3678.595} C_VEL
LIN {X 0,Y 545.413,Z 357.093,A -85,B 0,C 180,E1 -3679.419,E2 -3679.419} C_VEL
LIN {X 0,Y 545.166,Z 367.534,A -85,B 0,C 180,E1 -3680.352,E2 -3680.352} C_VEL
LIN {X 0,Y 545.027,Z 375.987,A -85,B 0,C 180,E1 -3681.285,E2 -3681.285} C_VEL
LIN {X 0,Y 544.861,Z 384.235,A -85,B 0,C 180,E1 -3682.402,E2 -3682.402} C_VEL
LIN {X 0,Y 544.735,Z 391.618,A -85,B 0,C 180,E1 -3683.655,E2 -3683.655} C_VEL
LIN {X 0,Y 544.654,Z 396.948,A -85,B 0,C 180,E1 -3684.817,E2 -3684.817} C_VEL
LIN {X 0,Y 544.684,Z 400.894,A -85,B 0,C 180,E1 -3685.93,E2 -3685.93} C_VEL
LIN {X 0,Y 544.651,Z 403.807,A -85,B 0,C 180,E1 -3687.041,E2 -3687.041} C_VEL
LIN {X 0,Y 544.546,Z 406.185,A -85,B 0,C 180,E1 -3688.52,E2 -3688.52} C_VEL
LIN {X 0,Y 544.541,Z 407,A -85,B 0,C 180,E1 -3690,E2 -3690} C_VEL
LIN {X 0,Y 544.546,Z 406.187,A -85,B 0,C 180,E1 -3691.479,E2 -3691.479} C_VEL
LIN {X 0,Y 544.651,Z 403.811,A -85,B 0,C 180,E1 -3692.958,E2 -3692.958} C_VEL
LIN {X 0,Y 544.684,Z 400.897,A -85,B 0,C 180,E1 -3694.069,E2 -3694.069} C_VEL
LIN {X 0,Y 544.654,Z 396.951,A -85,B 0,C 180,E1 -3695.182,E2 -3695.182} C_VEL
LIN {X 0,Y 544.735,Z 391.616,A -85,B 0,C 180,E1 -3696.345,E2 -3696.345} C_VEL
LIN {X 0,Y 544.86,Z 384.24,A -85,B 0,C 180,E1 -3697.597,E2 -3697.597} C_VEL
LIN {X 0,Y 545.029,Z 375.994,A -85,B 0,C 180,E1 -3698.714,E2 -3698.714} C_VEL
LIN {X 0,Y 545.165,Z 367.543,A -85,B 0,C 180,E1 -3699.647,E2 -3699.647} C_VEL
LIN {X 0,Y 545.412,Z 357.103,A -85,B 0,C 180,E1 -3700.58,E2 -3700.58} C_VEL
LIN {X 0,Y 545.618,Z 345.677,A -85,B 0,C 180,E1 -3701.4,E2 -3701.4} C_VEL
LIN {X 0,Y 545.768,Z 335.42,A -85,B 0,C 180,E1 -3701.984,E2 -3701.984} C_VEL
LIN {X 0,Y 545.951,Z 323.776,A -85,B 0,C 180,E1 -3702.499,E2 -3702.499} C_VEL
LIN {X 0,Y 546.137,Z 310.367,A -85,B 0,C 180,E1 -3702.92,E2 -3702.92} C_VEL
LIN {X 0,Y 545.734,Z 305.124,A -85,B 0,C 180,E1 -3703.05,E2 -3703.05} C_VEL
LIN {X 0,Y 544.803,Z 299.532,A -85,B 0,C 180,E1 -3703.189,E2 -3703.189} C_VEL
LIN {X 0,Y 544.937,Z 289.437,A -85,B 0,C 180,E1 -3706.098,E2 -3706.098} C_VEL
LIN {X 0,Y 545.068,Z 278.846,A -85,B 0,C 180,E1 -3709.195,E2 -3709.195} C_VEL
LIN {X 0,Y 545.218,Z 268.255,A -85,B 0,C 180,E1 -3712.349,E2 -3712.349} C_VEL
LIN {X 0,Y 545.357,Z 258.988,A -85,B 0,C 180,E1 -3715.167,E2 -3715.167} C_VEL
LIN {X 0,Y 545.559,Z 249.72,A -85,B 0,C 180,E1 -3718.047,E2 -3718.047} C_VEL
LIN {X 0,Y 545.711,Z 240.453,A -85,B 0,C 180,E1 -3721.006,E2 -3721.006} C_VEL
LIN {X 0,Y 545.931,Z 232.45,A -85,B 0,C 180,E1 -3723.611,E2 -3723.611} C_VEL
LIN {X 0,Y 545.93,Z 225.845,A -85,B 0,C 180,E1 -3725.803,E2 -3725.803} C_VEL
LIN {X 0,Y 545.069,Z 220.593,A -85,B 0,C 180,E1 -3727.812,E2 -3727.812} C_VEL
LIN {X 0,Y 545.082,Z 220.591,A -85,B 0,C 180,E1 -3730.472,E2 -3730.472} C_VEL
LIN {X 0,Y 545.079,Z 220.59,A -85,B 0,C 180,E1 -3733.106,E2 -3733.106} C_VEL
LIN {X 0,Y 545.068,Z 220.591,A -85,B 0,C 180,E1 -3736.223,E2 -3736.223} C_VEL
LIN {X 0,Y 545.102,Z 220.588,A -85,B 0,C 180,E1 -3738.886,E2 -3738.886} C_VEL
LIN {X 0,Y 545.055,Z 220.594,A -85,B 0,C 180,E1 -3741.762,E2 -3741.762} C_VEL
LIN {X 0,Y 545.037,Z 220.595,A -85,B 0,C 180,E1 -3744.531,E2 -3744.531} C_VEL
LIN {X 0,Y 545.068,Z 220.592,A -85,B 0,C 180,E1 -3747.211,E2 -3747.211} C_VEL
LIN {X 0,Y 545.065,Z 220.592,A -85,B 0,C 180,E1 -3749.81,E2 -3749.81} C_VEL
LIN {X 0,Y 545.094,Z 220.589,A -85,B 0,C 180,E1 -3752.344,E2 -3752.344} C_VEL
LIN {X 0,Y 545.118,Z 220.584,A -85,B 0,C 180,E1 -3754.819,E2 -3754.819} C_VEL
LIN {X 0,Y 545.044,Z 220.595,A -85,B 0,C 180,E1 -3757.242,E2 -3757.242} C_VEL
LIN {X 0,Y 545.12,Z 220.585,A -85,B 0,C 180,E1 -3760.414,E2 -3760.414} C_VEL
LIN {X 0,Y 545.075,Z 220.591,A -85,B 0,C 180,E1 -3763.52,E2 -3763.52} C_VEL
LIN {X 0,Y 545.094,Z 220.589,A -85,B 0,C 180,E1 -3765.819,E2 -3765.819} C_VEL
LIN {X 0,Y 545.115,Z 220.587,A -85,B 0,C 180,E1 -3768.848,E2 -3768.848} C_VEL
LIN {X 0,Y 545.129,Z 220.584,A -85,B 0,C 180,E1 -3771.846,E2 -3771.846} C_VEL
LIN {X 0,Y 545.204,Z 220.574,A -85,B 0,C 180,E1 -3774.822,E2 -3774.822} C_VEL
LIN {X 0,Y 545.192,Z 220.575,A -85,B 0,C 180,E1 -3777.782,E2 -3777.782} C_VEL
LIN {X 0,Y 545.212,Z 220.573,A -85,B 0,C 180,E1 -3780.737,E2 -3780.737} C_VEL
LIN {X 0,Y 545.17,Z 220.578,A -85,B 0,C 180,E1 -3782.955,E2 -3782.955} C_VEL
LIN {X 0,Y 545.166,Z 220.579,A -85,B 0,C 180,E1 -3785.918,E2 -3785.918} C_VEL
LIN {X 0,Y 545.123,Z 220.585,A -85,B 0,C 180,E1 -3788.899,E2 -3788.899} C_VEL
LIN {X 0,Y 545,Z 220.604,A -85,B 0,C 180,E1 -3791.906,E2 -3791.906} C_VEL
LIN {X 0,Y 544.849,Z 220.961,A -85,B 0,C 180,E1 -3793.424,E2 -3793.424} C_VEL
LIN {X 0,Y 544.842,Z 223.605,A -85,B 0,C 180,E1 -3795.715,E2 -3795.715} C_VEL
LIN {X 0,Y 544.819,Z 226.24,A -85,B 0,C 180,E1 -3798.033,E2 -3798.033} C_VEL
LIN {X 0,Y 544.773,Z 228.885,A -85,B 0,C 180,E1 -3800.383,E2 -3800.383} C_VEL
LIN {X 0,Y 544.75,Z 232.506,A -85,B 0,C 180,E1 -3803.654,E2 -3803.654} C_VEL
LIN {X 0,Y 544.717,Z 236.102,A -85,B 0,C 180,E1 -3806.843,E2 -3806.843} C_VEL
LIN {X 0,Y 544.626,Z 238.944,A -85,B 0,C 180,E1 -3809.362,E2 -3809.362} C_VEL
LIN {X 0,Y 544.577,Z 241.788,A -85,B 0,C 180,E1 -3811.944,E2 -3811.944} C_VEL
LIN {X 0,Y 544.609,Z 244.062,A -85,B 0,C 180,E1 -3813.94,E2 -3813.94} C_VEL
LIN {X 0,Y 546.109,Z 253.841,A -85,B 0,C 180,E1 -3814.211,E2 -3814.211} C_VEL
LIN {X 0,Y 545.961,Z 267.184,A -85,B 0,C 180,E1 -3814.679,E2 -3814.679} C_VEL
LIN {X 0,Y 545.851,Z 271.815,A -85,B 0,C 180,E1 -3814.882,E2 -3814.882} C_VEL
LIN {X 0,Y 545.022,Z 277.265,A -85,B 0,C 180,E1 -3815.132,E2 -3815.132} C_VEL
LIN {X 0,Y 542.003,Z 285.849,A -85,B 0,C 180,E1 -3815.56,E2 -3815.56} C_VEL
LIN {X 0,Y 539.077,Z 293.977,A -85,B 0,C 180,E1 -3816.059,E2 -3816.059} C_VEL
LIN {X 0,Y 538.371,Z 298.658,A -85,B 0,C 180,E1 -3816.417,E2 -3816.417} C_VEL
LIN {X 0,Y 538.155,Z 308.299,A -85,B 0,C 180,E1 -3817.311,E2 -3817.311} C_VEL
LIN {X 0,Y 537.918,Z 317.597,A -85,B 0,C 180,E1 -3818.381,E2 -3818.381} C_VEL
LIN {X 0,Y 537.797,Z 325.81,A -85,B 0,C 180,E1 -3819.555,E2 -3819.555} C_VEL
LIN {X 0,Y 537.65,Z 332.71,A -85,B 0,C 180,E1 -3820.81,E2 -3820.81} C_VEL
LIN {X 0,Y 537.608,Z 337.174,A -85,B 0,C 180,E1 -3821.829,E2 -3821.829} C_VEL
LIN {X 0,Y 537.571,Z 340.984,A -85,B 0,C 180,E1 -3822.936,E2 -3822.936} C_VEL
LIN {X 0,Y 537.521,Z 343.761,A -85,B 0,C 180,E1 -3824.019,E2 -3824.019} C_VEL
LIN {X 0,Y 537.492,Z 345.625,A -85,B 0,C 180,E1 -3825.084,E2 -3825.084} C_VEL
LIN {X 0,Y 537.464,Z 346.679,A -85,B 0,C 180,E1 -3826.13,E2 -3826.13} C_VEL
LIN {X 0,Y 537.452,Z 346.982,A -85,B 0,C 180,E1 -3827.159,E2 -3827.159} C_VEL
LIN {X 0,Y 537.464,Z 346.534,A -85,B 0,C 180,E1 -3828.186,E2 -3828.186} C_VEL
LIN {X 0,Y 537.459,Z 345.148,A -85,B 0,C 180,E1 -3829.323,E2 -3829.323} C_VEL
LIN {X 0,Y 537.501,Z 342.797,A -85,B 0,C 180,E1 -3830.481,E2 -3830.481} C_VEL
LIN {X 0,Y 537.555,Z 339.34,A -85,B 0,C 180,E1 -3831.666,E2 -3831.666} C_VEL
LIN {X 0,Y 537.631,Z 333.858,A -85,B 0,C 180,E1 -3833.036,E2 -3833.036} C_VEL
LIN {X 0,Y 537.756,Z 327.081,A -85,B 0,C 180,E1 -3834.32,E2 -3834.32} C_VEL
LIN {X 0,Y 537.885,Z 319.941,A -85,B 0,C 180,E1 -3835.399,E2 -3835.399} C_VEL
LIN {X 0,Y 538.106,Z 310.781,A -85,B 0,C 180,E1 -3836.51,E2 -3836.51} C_VEL
LIN {X 0,Y 538.313,Z 300.331,A -85,B 0,C 180,E1 -3837.527,E2 -3837.527} C_VEL
LIN {X 0,Y 538.567,Z 289.525,A -85,B 0,C 180,E1 -3838.366,E2 -3838.366} C_VEL
LIN {X 0,Y 538.808,Z 277.499,A -85,B 0,C 180,E1 -3839.098,E2 -3839.098} C_VEL
LIN {X 0,Y 539.051,Z 266.131,A -85,B 0,C 180,E1 -3839.63,E2 -3839.63} C_VEL
LIN {X 0,Y 539.161,Z 253.297,A -85,B 0,C 180,E1 -3840.069,E2 -3840.069} C_VEL
LIN {X 0,Y 537.529,Z 244.318,A -85,B 0,C 180,E1 -3840.344,E2 -3840.344} C_VEL
LIN {X 0,Y 537.568,Z 240.512,A -85,B 0,C 180,E1 -3843.609,E2 -3843.609} C_VEL
LIN {X 0,Y 537.599,Z 237.57,A -85,B 0,C 180,E1 -3846.216,E2 -3846.216} C_VEL
LIN {X 0,Y 537.614,Z 234.919,A -85,B 0,C 180,E1 -3848.529,E2 -3848.529} C_VEL
LIN {X 0,Y 537.644,Z 232.191,A -85,B 0,C 180,E1 -3850.926,E2 -3850.926} C_VEL
LIN {X 0,Y 537.661,Z 229.473,A -85,B 0,C 180,E1 -3853.288,E2 -3853.288} C_VEL
LIN {X 0,Y 537.718,Z 226.809,A -85,B 0,C 180,E1 -3855.622,E2 -3855.622} C_VEL
LIN {X 0,Y 537.832,Z 223.271,A -85,B 0,C 180,E1 -3858.697,E2 -3858.697} C_VEL
LIN {X 0,Y 537.722,Z 221.559,A -85,B 0,C 180,E1 -3860.218,E2 -3860.218} C_VEL
LIN {X 0,Y 538.113,Z 221.456,A -85,B 0,C 180,E1 -3863.005,E2 -3863.005} C_VEL
LIN {X 0,Y 538.172,Z 221.451,A -85,B 0,C 180,E1 -3864.756,E2 -3864.756} C_VEL
LIN {X 0,Y 538.153,Z 221.452,A -85,B 0,C 180,E1 -3867.755,E2 -3867.755} C_VEL
LIN {X 0,Y 538.174,Z 221.451,A -85,B 0,C 180,E1 -3870.749,E2 -3870.749} C_VEL
LIN {X 0,Y 538.127,Z 221.457,A -85,B 0,C 180,E1 -3872.995,E2 -3872.995} C_VEL
LIN {X 0,Y 538.111,Z 221.456,A -85,B 0,C 180,E1 -3875.998,E2 -3875.998} C_VEL
LIN {X 0,Y 538.062,Z 221.466,A -85,B 0,C 180,E1 -3879.018,E2 -3879.018} C_VEL
LIN {X 0,Y 538.069,Z 221.461,A -85,B 0,C 180,E1 -3882.063,E2 -3882.063} C_VEL
LIN {X 0,Y 538.031,Z 221.468,A -85,B 0,C 180,E1 -3885.145,E2 -3885.145} C_VEL
LIN {X 0,Y 538.023,Z 221.468,A -85,B 0,C 180,E1 -3888.271,E2 -3888.271} C_VEL
LIN {X 0,Y 538.029,Z 221.468,A -85,B 0,C 180,E1 -3890.652,E2 -3890.652} C_VEL
LIN {X 0,Y 538.03,Z 221.468,A -85,B 0,C 180,E1 -3893.071,E2 -3893.071} C_VEL
LIN {X 0,Y 538.039,Z 221.467,A -85,B 0,C 180,E1 -3895.676,E2 -3895.676} C_VEL
LIN {X 0,Y 538.036,Z 221.468,A -85,B 0,C 180,E1 -3898.05,E2 -3898.05} C_VEL
LIN {X 0,Y 538.007,Z 221.471,A -85,B 0,C 180,E1 -3900.628,E2 -3900.628} C_VEL
LIN {X 0,Y 538.032,Z 221.466,A -85,B 0,C 180,E1 -3903.284,E2 -3903.284} C_VEL
LIN {X 0,Y 538.015,Z 221.468,A -85,B 0,C 180,E1 -3906.003,E2 -3906.003} C_VEL
LIN {X 0,Y 538.005,Z 221.472,A -85,B 0,C 180,E1 -3908.831,E2 -3908.831} C_VEL
LIN {X 0,Y 538.049,Z 221.464,A -85,B 0,C 180,E1 -3911.772,E2 -3911.772} C_VEL
LIN {X 0,Y 538.023,Z 221.467,A -85,B 0,C 180,E1 -3915.142,E2 -3915.142} C_VEL
LIN {X 0,Y 538.032,Z 221.469,A -85,B 0,C 180,E1 -3918.229,E2 -3918.229} C_VEL
LIN {X 0,Y 538.052,Z 221.465,A -85,B 0,C 180,E1 -3920.413,E2 -3920.413} C_VEL
LIN {X 0,Y 538.022,Z 221.47,A -85,B 0,C 180,E1 -3923.069,E2 -3923.069} C_VEL
LIN {X 0,Y 538.024,Z 221.468,A -85,B 0,C 180,E1 -3925.829,E2 -3925.829} C_VEL
LIN {X 0,Y 538.019,Z 221.468,A -85,B 0,C 180,E1 -3928.501,E2 -3928.501} C_VEL
LIN {X 0,Y 538.055,Z 221.464,A -85,B 0,C 180,E1 -3931.101,E2 -3931.101} C_VEL
LIN {X 0,Y 538.038,Z 221.466,A -85,B 0,C 180,E1 -3933.635,E2 -3933.635} C_VEL
LIN {X 0,Y 538.02,Z 221.471,A -85,B 0,C 180,E1 -3936.12,E2 -3936.12} C_VEL
LIN {X 0,Y 538.037,Z 221.465,A -85,B 0,C 180,E1 -3939.35,E2 -3939.35} C_VEL
LIN {X 0,Y 538.072,Z 221.462,A -85,B 0,C 180,E1 -3942.519,E2 -3942.519} C_VEL
LIN {X 0,Y 538.063,Z 221.464,A -85,B 0,C 180,E1 -3945.632,E2 -3945.632} C_VEL
LIN {X 0,Y 538.078,Z 221.46,A -85,B 0,C 180,E1 -3948.703,E2 -3948.703} C_VEL
LIN {X 0,Y 538.059,Z 221.466,A -85,B 0,C 180,E1 -3951.741,E2 -3951.741} C_VEL
LIN {X 0,Y 538.125,Z 221.458,A -85,B 0,C 180,E1 -3954.004,E2 -3954.004} C_VEL
LIN {X 0,Y 538.139,Z 221.452,A -85,B 0,C 180,E1 -3957.007,E2 -3957.007} C_VEL
LIN {X 0,Y 538.176,Z 221.452,A -85,B 0,C 180,E1 -3960.001,E2 -3960.001} C_VEL
LIN {X 0,Y 538.139,Z 221.453,A -85,B 0,C 180,E1 -3962.996,E2 -3962.996} C_VEL
LIN {X 0,Y 538.117,Z 221.458,A -85,B 0,C 180,E1 -3965.999,E2 -3965.999} C_VEL
LIN {X 0,Y 538.058,Z 221.463,A -85,B 0,C 180,E1 -3969.019,E2 -3969.019} C_VEL
LIN {X 0,Y 538.087,Z 221.461,A -85,B 0,C 180,E1 -3972.064,E2 -3972.064} C_VEL
LIN {X 0,Y 538.05,Z 221.464,A -85,B 0,C 180,E1 -3975.145,E2 -3975.145} C_VEL
LIN {X 0,Y 538.036,Z 221.465,A -85,B 0,C 180,E1 -3978.271,E2 -3978.271} C_VEL
LIN {X 0,Y 538.042,Z 221.466,A -85,B 0,C 180,E1 -3980.652,E2 -3980.652} C_VEL
LIN {X 0,Y 538.012,Z 221.471,A -85,B 0,C 180,E1 -3983.878,E2 -3983.878} C_VEL
LIN {X 0,Y 538.042,Z 221.467,A -85,B 0,C 180,E1 -3986.368,E2 -3986.368} C_VEL
LIN {X 0,Y 538.036,Z 221.467,A -85,B 0,C 180,E1 -3988.934,E2 -3988.934} C_VEL
LIN {X 0,Y 538.015,Z 221.469,A -85,B 0,C 180,E1 -3991.888,E2 -3991.888} C_VEL
LIN {X 0,Y 538.015,Z 221.471,A -85,B 0,C 180,E1 -3994.618,E2 -3994.618} C_VEL
LIN {X 0,Y 538.01,Z 221.471,A -85,B 0,C 180,E1 -3997.17,E2 -3997.17} C_VEL
LIN {X 0,Y 538.028,Z 221.466,A -85,B 0,C 180,E1 -3999.797,E2 -3999.797} C_VEL
LIN {X 0,Y 538.025,Z 221.469,A -85,B 0,C 180,E1 -4002.786,E2 -4002.786} C_VEL
LIN {X 0,Y 538.025,Z 221.467,A -85,B 0,C 180,E1 -4005.927,E2 -4005.927} C_VEL
LIN {X 0,Y 538.036,Z 221.467,A -85,B 0,C 180,E1 -4008.227,E2 -4008.227} C_VEL
LIN {X 0,Y 538.019,Z 221.471,A -85,B 0,C 180,E1 -4011.17,E2 -4011.17} C_VEL
LIN {X 0,Y 538.044,Z 221.551,A -85,B 0,C 180,E1 -4011.998,E2 -4011.998} C_VEL
LIN {X 0,Y 539,Z 227.255,A -85,B 0,C 180,E1 -4014.073,E2 -4014.073} C_VEL
LIN {X 0,Y 538.95,Z 234.525,A -85,B 0,C 180,E1 -4016.572,E2 -4016.572} C_VEL
LIN {X 0,Y 538.726,Z 243.141,A -85,B 0,C 180,E1 -4019.431,E2 -4019.431} C_VEL
LIN {X 0,Y 538.502,Z 252.866,A -85,B 0,C 180,E1 -4022.558,E2 -4022.558} C_VEL
LIN {X 0,Y 538.34,Z 261.633,A -85,B 0,C 180,E1 -4025.307,E2 -4025.307} C_VEL
LIN {X 0,Y 538.18,Z 270.408,A -85,B 0,C 180,E1 -4028,E2 -4028} C_VEL
LIN {X 0,Y 538.027,Z 278.843,A -85,B 0,C 180,E1 -4030.543,E2 -4030.543} C_VEL
LIN {X 0,Y 537.895,Z 288.11,A -85,B 0,C 180,E1 -4033.295,E2 -4033.295} C_VEL
LIN {X 0,Y 537.779,Z 297.378,A -85,B 0,C 180,E1 -4036.009,E2 -4036.009} C_VEL
LIN {X 0,Y 537.736,Z 299.529,A -85,B 0,C 180,E1 -4036.634,E2 -4036.634} C_VEL
LIN {X 0,Y 539.252,Z 310.339,A -85,B 0,C 180,E1 -4036.912,E2 -4036.912} C_VEL
LIN {X 0,Y 539.042,Z 322.465,A -85,B 0,C 180,E1 -4037.29,E2 -4037.29} C_VEL
LIN {X 0,Y 538.84,Z 333.48,A -85,B 0,C 180,E1 -4037.763,E2 -4037.763} C_VEL
LIN {X 0,Y 538.652,Z 344.426,A -85,B 0,C 180,E1 -4038.372,E2 -4038.372} C_VEL
LIN {X 0,Y 538.429,Z 355.921,A -85,B 0,C 180,E1 -4039.185,E2 -4039.185} C_VEL
LIN {X 0,Y 538.202,Z 365.598,A -85,B 0,C 180,E1 -4040.036,E2 -4040.036} C_VEL
LIN {X 0,Y 538.015,Z 374.41,A -85,B 0,C 180,E1 -4040.981,E2 -4040.981} C_VEL
LIN {X 0,Y 537.831,Z 382.999,A -85,B 0,C 180,E1 -4042.113,E2 -4042.113} C_VEL
LIN {X 0,Y 537.707,Z 389.866,A -85,B 0,C 180,E1 -4043.244,E2 -4043.244} C_VEL
LIN {X 0,Y 537.677,Z 395.364,A -85,B 0,C 180,E1 -4044.374,E2 -4044.374} C_VEL
LIN {X 0,Y 537.558,Z 399.676,A -85,B 0,C 180,E1 -4045.5,E2 -4045.5} C_VEL
LIN {X 0,Y 537.592,Z 401.956,A -85,B 0,C 180,E1 -4046.252,E2 -4046.252} C_VEL
LIN {X 0,Y 537.552,Z 403.807,A -85,B 0,C 180,E1 -4047.002,E2 -4047.002} C_VEL
LIN {X 0,Y 537.49,Z 405.197,A -85,B 0,C 180,E1 -4047.751,E2 -4047.751} C_VEL
LIN {X 0,Y 537.442,Z 406.785,A -85,B 0,C 180,E1 -4049.25,E2 -4049.25} C_VEL
LIN {X 0,Y 537.442,Z 407,A -85,B 0,C 180,E1 -4050,E2 -4050} C_VEL
LIN {X 0,Y 537.452,Z 406.187,A -85,B 0,C 180,E1 -4051.498,E2 -4051.498} C_VEL
LIN {X 0,Y 537.49,Z 405.2,A -85,B 0,C 180,E1 -4052.248,E2 -4052.248} C_VEL
LIN {X 0,Y 537.551,Z 403.811,A -85,B 0,C 180,E1 -4052.997,E2 -4052.997} C_VEL
LIN {X 0,Y 537.604,Z 400.897,A -85,B 0,C 180,E1 -4054.123,E2 -4054.123} C_VEL
LIN {X 0,Y 537.588,Z 396.951,A -85,B 0,C 180,E1 -4055.25,E2 -4055.25} C_VEL
LIN {X 0,Y 537.65,Z 392.104,A -85,B 0,C 180,E1 -4056.33,E2 -4056.33} C_VEL
LIN {X 0,Y 537.791,Z 385.472,A -85,B 0,C 180,E1 -4057.509,E2 -4057.509} C_VEL
LIN {X 0,Y 537.973,Z 377.482,A -85,B 0,C 180,E1 -4058.64,E2 -4058.64} C_VEL
LIN {X 0,Y 538.119,Z 369.34,A -85,B 0,C 180,E1 -4059.585,E2 -4059.585} C_VEL
LIN {X 0,Y 538.342,Z 359.406,A -85,B 0,C 180,E1 -4060.531,E2 -4060.531} C_VEL
LIN {X 0,Y 538.547,Z 349.594,A -85,B 0,C 180,E1 -4061.288,E2 -4061.288} C_VEL
LIN {X 0,Y 538.714,Z 338.627,A -85,B 0,C 180,E1 -4061.969,E2 -4061.969} C_VEL
LIN {X 0,Y 538.986,Z 326.121,A -85,B 0,C 180,E1 -4062.567,E2 -4062.567} C_VEL
LIN {X 0,Y 539.18,Z 313.108,A -85,B 0,C 180,E1 -4063.017,E2 -4063.017} C_VEL
LIN {X 0,Y 539.005,Z 307.103,A -85,B 0,C 180,E1 -4063.174,E2 -4063.174} C_VEL
LIN {X 0,Y 537.736,Z 299.532,A -85,B 0,C 180,E1 -4063.365,E2 -4063.365} C_VEL
LIN {X 0,Y 537.877,Z 289.437,A -85,B 0,C 180,E1 -4066.315,E2 -4066.315} C_VEL
LIN {X 0,Y 537.996,Z 280.17,A -85,B 0,C 180,E1 -4069.061,E2 -4069.061} C_VEL
LIN {X 0,Y 538.127,Z 272.227,A -85,B 0,C 180,E1 -4071.449,E2 -4071.449} C_VEL
LIN {X 0,Y 538.324,Z 262.961,A -85,B 0,C 180,E1 -4074.282,E2 -4074.282} C_VEL
LIN {X 0,Y 538.483,Z 253.692,A -85,B 0,C 180,E1 -4077.18,E2 -4077.18} C_VEL
LIN {X 0,Y 538.7,Z 244.446,A -85,B 0,C 180,E1 -4080.143,E2 -4080.143} C_VEL
LIN {X 0,Y 538.894,Z 235.054,A -85,B 0,C 180,E1 -4083.212,E2 -4083.212} C_VEL
LIN {X 0,Y 539.026,Z 228.299,A -85,B 0,C 180,E1 -4085.464,E2 -4085.464} C_VEL
LIN {X 0,Y 538.439,Z 223.549,A -85,B 0,C 180,E1 -4087.23,E2 -4087.23} C_VEL
LIN {X 0,Y 538.026,Z 221.47,A -85,B 0,C 180,E1 -4088.071,E2 -4088.071} C_VEL
LIN {X 0,Y 538.049,Z 221.466,A -85,B 0,C 180,E1 -4090.775,E2 -4090.775} C_VEL
LIN {X 0,Y 538.031,Z 221.468,A -85,B 0,C 180,E1 -4094.074,E2 -4094.074} C_VEL
LIN {X 0,Y 538.027,Z 221.468,A -85,B 0,C 180,E1 -4097.012,E2 -4097.012} C_VEL
LIN {X 0,Y 538.08,Z 221.462,A -85,B 0,C 180,E1 -4099.248,E2 -4099.248} C_VEL
LIN {X 0,Y 537.994,Z 221.473,A -85,B 0,C 180,E1 -4102.121,E2 -4102.121} C_VEL
LIN {X 0,Y 537.999,Z 221.473,A -85,B 0,C 180,E1 -4104.915,E2 -4104.915} C_VEL
LIN {X 0,Y 538.018,Z 221.469,A -85,B 0,C 180,E1 -4107.616,E2 -4107.616} C_VEL
LIN {X 0,Y 538.017,Z 221.47,A -85,B 0,C 180,E1 -4110.238,E2 -4110.238} C_VEL
LIN {X 0,Y 538.07,Z 221.463,A -85,B 0,C 180,E1 -4112.796,E2 -4112.796} C_VEL
LIN {X 0,Y 538.049,Z 221.467,A -85,B 0,C 180,E1 -4115.292,E2 -4115.292} C_VEL
LIN {X 0,Y 538.014,Z 221.469,A -85,B 0,C 180,E1 -4118.041,E2 -4118.041} C_VEL
LIN {X 0,Y 538.037,Z 221.466,A -85,B 0,C 180,E1 -4120.939,E2 -4120.939} C_VEL
LIN {X 0,Y 538.025,Z 221.468,A -85,B 0,C 180,E1 -4123.298,E2 -4123.298} C_VEL
LIN {X 0,Y 538.062,Z 221.465,A -85,B 0,C 180,E1 -4125.63,E2 -4125.63} C_VEL
LIN {X 0,Y 538.074,Z 221.463,A -85,B 0,C 180,E1 -4128.7,E2 -4128.7} C_VEL
LIN {X 0,Y 538.085,Z 221.46,A -85,B 0,C 180,E1 -4131.738,E2 -4131.738} C_VEL
LIN {X 0,Y 538.161,Z 221.451,A -85,B 0,C 180,E1 -4134.754,E2 -4134.754} C_VEL
LIN {X 0,Y 538.164,Z 221.45,A -85,B 0,C 180,E1 -4137.753,E2 -4137.753} C_VEL
LIN {X 0,Y 538.182,Z 221.449,A -85,B 0,C 180,E1 -4140.747,E2 -4140.747} C_VEL
LIN {X 0,Y 538.136,Z 221.454,A -85,B 0,C 180,E1 -4142.993,E2 -4142.993} C_VEL
LIN {X 0,Y 538.119,Z 221.457,A -85,B 0,C 180,E1 -4145.996,E2 -4145.996} C_VEL
LIN {X 0,Y 538.072,Z 221.463,A -85,B 0,C 180,E1 -4149.016,E2 -4149.016} C_VEL
LIN {X 0,Y 538.012,Z 221.472,A -85,B 0,C 180,E1 -4151.563,E2 -4151.563} C_VEL
LIN {X 0,Y 537.849,Z 221.493,A -85,B 0,C 180,E1 -4152.833,E2 -4152.833} C_VEL
LIN {X 0,Y 537.793,Z 221.939,A -85,B 0,C 180,E1 -4153.604,E2 -4153.604} C_VEL
LIN {X 0,Y 537.784,Z 224.578,A -85,B 0,C 180,E1 -4155.927,E2 -4155.927} C_VEL
LIN {X 0,Y 537.757,Z 227.209,A -85,B 0,C 180,E1 -4158.278,E2 -4158.278} C_VEL
LIN {X 0,Y 537.698,Z 229.872,A -85,B 0,C 180,E1 -4160.663,E2 -4160.663} C_VEL
LIN {X 0,Y 537.683,Z 233.496,A -85,B 0,C 180,E1 -4163.902,E2 -4163.902} C_VEL
LIN {X 0,Y 537.62,Z 236.241,A -85,B 0,C 180,E1 -4166.387,E2 -4166.387} C_VEL
LIN {X 0,Y 537.559,Z 239.115,A -85,B 0,C 180,E1 -4168.928,E2 -4168.928} C_VEL
LIN {X 0,Y 537.516,Z 242.258,A -85,B 0,C 180,E1 -4171.804,E2 -4171.804} C_VEL
LIN {X 0,Y 537.53,Z 244.484,A -85,B 0,C 180,E1 -4173.755,E2 -4173.755} C_VEL
LIN {X 0,Y 539.218,Z 254.597,A -85,B 0,C 180,E1 -4174.057,E2 -4174.057} C_VEL
LIN {X 0,Y 539.022,Z 267.199,A -85,B 0,C 180,E1 -4174.502,E2 -4174.502} C_VEL
LIN {X 0,Y 538.761,Z 279.242,A -85,B 0,C 180,E1 -4175.082,E2 -4175.082} C_VEL
LIN {X 0,Y 538.51,Z 290.923,A -85,B 0,C 180,E1 -4175.818,E2 -4175.818} C_VEL
LIN {X 0,Y 538.371,Z 298.658,A -85,B 0,C 180,E1 -4176.417,E2 -4176.417} C_VEL
LIN {X 0,Y 537.664,Z 303.293,A -85,B 0,C 180,E1 -4176.8,E2 -4176.8} C_VEL
LIN {X 0,Y 534.701,Z 310.544,A -85,B 0,C 180,E1 -4177.451,E2 -4177.451} C_VEL
LIN {X 0,Y 531.674,Z 317.215,A -85,B 0,C 180,E1 -4178.171,E2 -4178.171} C_VEL
LIN {X 0,Y 530.878,Z 320.941,A -85,B 0,C 180,E1 -4178.659,E2 -4178.659} C_VEL
LIN {X 0,Y 530.677,Z 328.355,A -85,B 0,C 180,E1 -4179.816,E2 -4179.816} C_VEL
LIN {X 0,Y 530.56,Z 334.292,A -85,B 0,C 180,E1 -4180.972,E2 -4180.972} C_VEL
LIN {X 0,Y 530.51,Z 338.903,A -85,B 0,C 180,E1 -4182.11,E2 -4182.11} C_VEL
LIN {X 0,Y 530.484,Z 342.374,A -85,B 0,C 180,E1 -4183.227,E2 -4183.227} C_VEL
LIN {X 0,Y 530.419,Z 345.381,A -85,B 0,C 180,E1 -4184.605,E2 -4184.605} C_VEL
LIN {X 0,Y 530.407,Z 346.759,A -85,B 0,C 180,E1 -4185.682,E2 -4185.682} C_VEL
LIN {X 0,Y 530.343,Z 347.358,A -85,B 0,C 180,E1 -4186.787,E2 -4186.787} C_VEL
LIN {X 0,Y 530.365,Z 347.126,A -85,B 0,C 180,E1 -4187.905,E2 -4187.905} C_VEL
LIN {X 0,Y 530.389,Z 346.015,A -85,B 0,C 180,E1 -4189.048,E2 -4189.048} C_VEL
LIN {X 0,Y 530.421,Z 343.264,A -85,B 0,C 180,E1 -4190.507,E2 -4190.507} C_VEL
LIN {X 0,Y 530.5,Z 338.899,A -85,B 0,C 180,E1 -4191.974,E2 -4191.974} C_VEL
LIN {X 0,Y 530.584,Z 334.684,A -85,B 0,C 180,E1 -4193.026,E2 -4193.026} C_VEL
LIN {X 0,Y 530.719,Z 327.795,A -85,B 0,C 180,E1 -4194.362,E2 -4194.362} C_VEL
LIN {X 0,Y 530.892,Z 320.156,A -85,B 0,C 180,E1 -4195.534,E2 -4195.534} C_VEL
LIN {X 0,Y 531.103,Z 311.956,A -85,B 0,C 180,E1 -4196.549,E2 -4196.549} C_VEL
LIN {X 0,Y 531.336,Z 302.224,A -85,B 0,C 180,E1 -4197.528,E2 -4197.528} C_VEL
LIN {X 0,Y 531.576,Z 291.395,A -85,B 0,C 180,E1 -4198.408,E2 -4198.408} C_VEL
LIN {X 0,Y 531.843,Z 280.265,A -85,B 0,C 180,E1 -4199.124,E2 -4199.124} C_VEL
LIN {X 0,Y 532.083,Z 268.34,A -85,B 0,C 180,E1 -4199.716,E2 -4199.716} C_VEL
LIN {X 0,Y 532.306,Z 255.385,A -85,B 0,C 180,E1 -4200.188,E2 -4200.188} C_VEL
LIN {X 0,Y 530.449,Z 244.744,A -85,B 0,C 180,E1 -4200.51,E2 -4200.51} C_VEL
LIN {X 0,Y 530.478,Z 241.611,A -85,B 0,C 180,E1 -4203.228,E2 -4203.228} C_VEL
LIN {X 0,Y 530.527,Z 238.35,A -85,B 0,C 180,E1 -4206.067,E2 -4206.067} C_VEL
LIN {X 0,Y 530.531,Z 234.954,A -85,B 0,C 180,E1 -4209.043,E2 -4209.043} C_VEL
LIN {X 0,Y 530.548,Z 232.199,A -85,B 0,C 180,E1 -4211.463,E2 -4211.463} C_VEL
LIN {X 0,Y 530.594,Z 229.469,A -85,B 0,C 180,E1 -4213.85,E2 -4213.85} C_VEL
LIN {X 0,Y 530.625,Z 226.782,A -85,B 0,C 180,E1 -4216.208,E2 -4216.208} C_VEL
LIN {X 0,Y 530.744,Z 223.242,A -85,B 0,C 180,E1 -4219.317,E2 -4219.317} C_VEL
LIN {X 0,Y 530.66,Z 222.388,A -85,B 0,C 180,E1 -4220.086,E2 -4220.086} C_VEL
LIN {X 0,Y 530.988,Z 222.345,A -85,B 0,C 180,E1 -4222.395,E2 -4222.395} C_VEL
LIN {X 0,Y 531.127,Z 222.328,A -85,B 0,C 180,E1 -4224.686,E2 -4224.686} C_VEL
LIN {X 0,Y 531.125,Z 222.327,A -85,B 0,C 180,E1 -4227.725,E2 -4227.725} C_VEL
LIN {X 0,Y 531.143,Z 222.327,A -85,B 0,C 180,E1 -4230.759,E2 -4230.759} C_VEL
LIN {X 0,Y 531.093,Z 222.334,A -85,B 0,C 180,E1 -4233.035,E2 -4233.035} C_VEL
LIN {X 0,Y 531.07,Z 222.333,A -85,B 0,C 180,E1 -4236.078,E2 -4236.078} C_VEL
LIN {X 0,Y 531.021,Z 222.342,A -85,B 0,C 180,E1 -4239.139,E2 -4239.139} C_VEL
LIN {X 0,Y 531.026,Z 222.339,A -85,B 0,C 180,E1 -4242.226,E2 -4242.226} C_VEL
LIN {X 0,Y 530.982,Z 222.345,A -85,B 0,C 180,E1 -4245.351,E2 -4245.351} C_VEL
LIN {X 0,Y 531.002,Z 222.341,A -85,B 0,C 180,E1 -4247.723,E2 -4247.723} C_VEL
LIN {X 0,Y 530.991,Z 222.346,A -85,B 0,C 180,E1 -4250.939,E2 -4250.939} C_VEL
LIN {X 0,Y 530.994,Z 222.342,A -85,B 0,C 180,E1 -4254.046,E2 -4254.046} C_VEL
LIN {X 0,Y 530.999,Z 222.345,A -85,B 0,C 180,E1 -4256.744,E2 -4256.744} C_VEL
LIN {X 0,Y 530.97,Z 222.347,A -85,B 0,C 180,E1 -4259.324,E2 -4259.324} C_VEL
LIN {X 0,Y 530.968,Z 222.346,A -85,B 0,C 180,E1 -4262.104,E2 -4262.104} C_VEL
LIN {X 0,Y 530.978,Z 222.346,A -85,B 0,C 180,E1 -4264.856,E2 -4264.856} C_VEL
LIN {X 0,Y 530.955,Z 222.35,A -85,B 0,C 180,E1 -4267.509,E2 -4267.509} C_VEL
LIN {X 0,Y 531.017,Z 222.341,A -85,B 0,C 180,E1 -4270.43,E2 -4270.43} C_VEL
LIN {X 0,Y 530.958,Z 222.349,A -85,B 0,C 180,E1 -4273.496,E2 -4273.496} C_VEL
LIN {X 0,Y 530.957,Z 222.348,A -85,B 0,C 180,E1 -4276.507,E2 -4276.507} C_VEL
LIN {X 0,Y 531.018,Z 222.342,A -85,B 0,C 180,E1 -4279.573,E2 -4279.573} C_VEL
LIN {X 0,Y 530.962,Z 222.348,A -85,B 0,C 180,E1 -4282.578,E2 -4282.578} C_VEL
LIN {X 0,Y 530.994,Z 222.345,A -85,B 0,C 180,E1 -4285.313,E2 -4285.313} C_VEL
LIN {X 0,Y 530.977,Z 222.347,A -85,B 0,C 180,E1 -4288.035,E2 -4288.035} C_VEL
LIN {X 0,Y 531.003,Z 222.342,A -85,B 0,C 180,E1 -4290.872,E2 -4290.872} C_VEL
LIN {X 0,Y 531.001,Z 222.341,A -85,B 0,C 180,E1 -4293.258,E2 -4293.258} C_VEL
LIN {X 0,Y 530.994,Z 222.344,A -85,B 0,C 180,E1 -4295.959,E2 -4295.959} C_VEL
LIN {X 0,Y 530.997,Z 222.342,A -85,B 0,C 180,E1 -4299.064,E2 -4299.064} C_VEL
LIN {X 0,Y 531.016,Z 222.342,A -85,B 0,C 180,E1 -4302.279,E2 -4302.279} C_VEL
LIN {X 0,Y 531.018,Z 222.34,A -85,B 0,C 180,E1 -4305.437,E2 -4305.437} C_VEL
LIN {X 0,Y 531.037,Z 222.337,A -85,B 0,C 180,E1 -4308.551,E2 -4308.551} C_VEL
LIN {X 0,Y 531.034,Z 222.34,A -85,B 0,C 180,E1 -4311.631,E2 -4311.631} C_VEL
LIN {X 0,Y 531.122,Z 222.326,A -85,B 0,C 180,E1 -4314.687,E2 -4314.687} C_VEL
LIN {X 0,Y 531.137,Z 222.328,A -85,B 0,C 180,E1 -4317.726,E2 -4317.726} C_VEL
LIN {X 0,Y 531.153,Z 222.323,A -85,B 0,C 180,E1 -4320.759,E2 -4320.759} C_VEL
LIN {X 0,Y 531.106,Z 222.329,A -85,B 0,C 180,E1 -4323.035,E2 -4323.035} C_VEL
LIN {X 0,Y 531.072,Z 222.335,A -85,B 0,C 180,E1 -4326.078,E2 -4326.078} C_VEL
LIN {X 0,Y 531.02,Z 222.34,A -85,B 0,C 180,E1 -4329.139,E2 -4329.139} C_VEL
LIN {X 0,Y 531.044,Z 222.337,A -85,B 0,C 180,E1 -4332.226,E2 -4332.226} C_VEL
LIN {X 0,Y 531,Z 222.344,A -85,B 0,C 180,E1 -4335.351,E2 -4335.351} C_VEL
LIN {X 0,Y 530.995,Z 222.342,A -85,B 0,C 180,E1 -4338.522,E2 -4338.522} C_VEL
LIN {X 0,Y 531.004,Z 222.342,A -85,B 0,C 180,E1 -4340.939,E2 -4340.939} C_VEL
LIN {X 0,Y 530.96,Z 222.347,A -85,B 0,C 180,E1 -4344.226,E2 -4344.226} C_VEL
LIN {X 0,Y 531.007,Z 222.342,A -85,B 0,C 180,E1 -4346.745,E2 -4346.745} C_VEL
LIN {X 0,Y 530.986,Z 222.345,A -85,B 0,C 180,E1 -4349.323,E2 -4349.323} C_VEL
LIN {X 0,Y 530.97,Z 222.348,A -85,B 0,C 180,E1 -4352.101,E2 -4352.101} C_VEL
LIN {X 0,Y 530.974,Z 222.347,A -85,B 0,C 180,E1 -4354.851,E2 -4354.851} C_VEL
LIN {X 0,Y 530.971,Z 222.346,A -85,B 0,C 180,E1 -4357.508,E2 -4357.508} C_VEL
LIN {X 0,Y 530.987,Z 222.346,A -85,B 0,C 180,E1 -4360.433,E2 -4360.433} C_VEL
LIN {X 0,Y 530.967,Z 222.346,A -85,B 0,C 180,E1 -4363.281,E2 -4363.281} C_VEL
LIN {X 0,Y 530.983,Z 222.345,A -85,B 0,C 180,E1 -4365.622,E2 -4365.622} C_VEL
LIN {X 0,Y 530.999,Z 222.344,A -85,B 0,C 180,E1 -4368.565,E2 -4368.565} C_VEL
LIN {X 0,Y 530.975,Z 222.346,A -85,B 0,C 180,E1 -4371.682,E2 -4371.682} C_VEL
LIN {X 0,Y 532.053,Z 228.765,A -85,B 0,C 180,E1 -4374.091,E2 -4374.091} C_VEL
LIN {X 0,Y 532.015,Z 235.273,A -85,B 0,C 180,E1 -4376.33,E2 -4376.33} C_VEL
LIN {X 0,Y 531.767,Z 243.821,A -85,B 0,C 180,E1 -4379.212,E2 -4379.212} C_VEL
LIN {X 0,Y 531.529,Z 253.689,A -85,B 0,C 180,E1 -4382.433,E2 -4382.433} C_VEL
LIN {X 0,Y 531.328,Z 262.956,A -85,B 0,C 180,E1 -4385.376,E2 -4385.376} C_VEL
LIN {X 0,Y 531.119,Z 272.224,A -85,B 0,C 180,E1 -4388.253,E2 -4388.253} C_VEL
LIN {X 0,Y 530.961,Z 281.491,A -85,B 0,C 180,E1 -4391.077,E2 -4391.077} C_VEL
LIN {X 0,Y 530.817,Z 290.758,A -85,B 0,C 180,E1 -4393.856,E2 -4393.856} C_VEL
LIN {X 0,Y 530.695,Z 299.529,A -85,B 0,C 180,E1 -4396.453,E2 -4396.453} C_VEL
LIN {X 0,Y 532.351,Z 310.339,A -85,B 0,C 180,E1 -4396.739,E2 -4396.739} C_VEL
LIN {X 0,Y 532.11,Z 323.76,A -85,B 0,C 180,E1 -4397.17,E2 -4397.17} C_VEL
LIN {X 0,Y 531.861,Z 335.404,A -85,B 0,C 180,E1 -4397.697,E2 -4397.697} C_VEL
LIN {X 0,Y 531.654,Z 346.302,A -85,B 0,C 180,E1 -4398.339,E2 -4398.339} C_VEL
LIN {X 0,Y 531.415,Z 357.094,A -85,B 0,C 180,E1 -4399.137,E2 -4399.137} C_VEL
LIN {X 0,Y 531.115,Z 367.535,A -85,B 0,C 180,E1 -4400.094,E2 -4400.094} C_VEL
LIN {X 0,Y 530.931,Z 375.988,A -85,B 0,C 180,E1 -4401.052,E2 -4401.052} C_VEL
LIN {X 0,Y 530.76,Z 384.235,A -85,B 0,C 180,E1 -4402.199,E2 -4402.199} C_VEL
LIN {X 0,Y 530.599,Z 391.271,A -85,B 0,C 180,E1 -4403.419,E2 -4403.419} C_VEL
LIN {X 0,Y 530.525,Z 396.948,A -85,B 0,C 180,E1 -4404.679,E2 -4404.679} C_VEL
LIN {X 0,Y 530.523,Z 400.894,A -85,B 0,C 180,E1 -4405.821,E2 -4405.821} C_VEL
LIN {X 0,Y 530.457,Z 403.807,A -85,B 0,C 180,E1 -4406.962,E2 -4406.962} C_VEL
LIN {X 0,Y 530.412,Z 405.197,A -85,B 0,C 180,E1 -4407.721,E2 -4407.721} C_VEL
LIN {X 0,Y 530.344,Z 406.785,A -85,B 0,C 180,E1 -4409.24,E2 -4409.24} C_VEL
LIN {X 0,Y 530.343,Z 407,A -85,B 0,C 180,E1 -4410,E2 -4410} C_VEL
LIN {X 0,Y 530.361,Z 406.186,A -85,B 0,C 180,E1 -4411.518,E2 -4411.518} C_VEL
LIN {X 0,Y 530.412,Z 405.2,A -85,B 0,C 180,E1 -4412.278,E2 -4412.278} C_VEL
LIN {X 0,Y 530.457,Z 403.811,A -85,B 0,C 180,E1 -4413.037,E2 -4413.037} C_VEL
LIN {X 0,Y 530.523,Z 400.897,A -85,B 0,C 180,E1 -4414.178,E2 -4414.178} C_VEL
LIN {X 0,Y 530.525,Z 396.95,A -85,B 0,C 180,E1 -4415.32,E2 -4415.32} C_VEL
LIN {X 0,Y 530.599,Z 391.272,A -85,B 0,C 180,E1 -4416.58,E2 -4416.58} C_VEL
LIN {X 0,Y 530.759,Z 384.24,A -85,B 0,C 180,E1 -4417.8,E2 -4417.8} C_VEL
LIN {X 0,Y 530.931,Z 375.994,A -85,B 0,C 180,E1 -4418.947,E2 -4418.947} C_VEL
LIN {X 0,Y 531.114,Z 367.543,A -85,B 0,C 180,E1 -4419.905,E2 -4419.905} C_VEL
LIN {X 0,Y 531.408,Z 357.104,A -85,B 0,C 180,E1 -4420.862,E2 -4420.862} C_VEL
LIN {X 0,Y 531.634,Z 345.361,A -85,B 0,C 180,E1 -4421.725,E2 -4421.725} C_VEL
LIN {X 0,Y 531.908,Z 333.496,A -85,B 0,C 180,E1 -4422.398,E2 -4422.398} C_VEL
LIN {X 0,Y 532.17,Z 321.183,A -85,B 0,C 180,E1 -4422.925,E2 -4422.925} C_VEL
LIN {X 0,Y 532.174,Z 308.537,A -85,B 0,C 180,E1 -4423.313,E2 -4423.313} C_VEL
LIN {X 0,Y 530.694,Z 299.532,A -85,B 0,C 180,E1 -4423.546,E2 -4423.546} C_VEL
LIN {X 0,Y 530.815,Z 290.761,A -85,B 0,C 180,E1 -4426.143,E2 -4426.143} C_VEL
LIN {X 0,Y 530.959,Z 281.494,A -85,B 0,C 180,E1 -4428.922,E2 -4428.922} C_VEL
LIN {X 0,Y 531.117,Z 272.227,A -85,B 0,C 180,E1 -4431.746,E2 -4431.746} C_VEL
LIN {X 0,Y 531.325,Z 262.959,A -85,B 0,C 180,E1 -4434.623,E2 -4434.623} C_VEL
LIN {X 0,Y 531.52,Z 253.477,A -85,B 0,C 180,E1 -4437.636,E2 -4437.636} C_VEL
LIN {X 0,Y 531.749,Z 243.794,A -85,B 0,C 180,E1 -4440.784,E2 -4440.784} C_VEL
LIN {X 0,Y 531.983,Z 234.959,A -85,B 0,C 180,E1 -4443.7,E2 -4443.7} C_VEL
LIN {X 0,Y 532.083,Z 229.553,A -85,B 0,C 180,E1 -4445.532,E2 -4445.532} C_VEL
LIN {X 0,Y 531.372,Z 224.474,A -85,B 0,C 180,E1 -4447.479,E2 -4447.479} C_VEL
LIN {X 0,Y 530.981,Z 222.348,A -85,B 0,C 180,E1 -4448.347,E2 -4448.347} C_VEL
LIN {X 0,Y 530.995,Z 222.347,A -85,B 0,C 180,E1 -4451.435,E2 -4451.435} C_VEL
LIN {X 0,Y 530.989,Z 222.347,A -85,B 0,C 180,E1 -4454.546,E2 -4454.546} C_VEL
LIN {X 0,Y 530.988,Z 222.346,A -85,B 0,C 180,E1 -4457.833,E2 -4457.833} C_VEL
LIN {X 0,Y 531.007,Z 222.343,A -85,B 0,C 180,E1 -4460.557,E2 -4460.557} C_VEL
LIN {X 0,Y 530.955,Z 222.349,A -85,B 0,C 180,E1 -4463.441,E2 -4463.441} C_VEL
LIN {X 0,Y 530.998,Z 222.344,A -85,B 0,C 180,E1 -4466.493,E2 -4466.493} C_VEL
LIN {X 0,Y 530.974,Z 222.347,A -85,B 0,C 180,E1 -4469.354,E2 -4469.354} C_VEL
LIN {X 0,Y 531.017,Z 222.342,A -85,B 0,C 180,E1 -4472.465,E2 -4472.465} C_VEL
LIN {X 0,Y 531.008,Z 222.342,A -85,B 0,C 180,E1 -4474.942,E2 -4474.942} C_VEL
LIN {X 0,Y 530.971,Z 222.347,A -85,B 0,C 180,E1 -4478.246,E2 -4478.246} C_VEL
LIN {X 0,Y 530.995,Z 222.345,A -85,B 0,C 180,E1 -4480.676,E2 -4480.676} C_VEL
LIN {X 0,Y 530.986,Z 222.345,A -85,B 0,C 180,E1 -4483.07,E2 -4483.07} C_VEL
LIN {X 0,Y 531.017,Z 222.341,A -85,B 0,C 180,E1 -4485.435,E2 -4485.435} C_VEL
LIN {X 0,Y 531.034,Z 222.339,A -85,B 0,C 180,E1 -4488.549,E2 -4488.549} C_VEL
LIN {X 0,Y 531.054,Z 222.335,A -85,B 0,C 180,E1 -4491.628,E2 -4491.628} C_VEL
LIN {X 0,Y 531.12,Z 222.328,A -85,B 0,C 180,E1 -4494.684,E2 -4494.684} C_VEL
LIN {X 0,Y 531.136,Z 222.325,A -85,B 0,C 180,E1 -4497.724,E2 -4497.724} C_VEL
LIN {X 0,Y 531.152,Z 222.324,A -85,B 0,C 180,E1 -4500.757,E2 -4500.757} C_VEL
LIN {X 0,Y 531.103,Z 222.33,A -85,B 0,C 180,E1 -4503.033,E2 -4503.033} C_VEL
LIN {X 0,Y 531.079,Z 222.334,A -85,B 0,C 180,E1 -4506.076,E2 -4506.076} C_VEL
LIN {X 0,Y 531.031,Z 222.34,A -85,B 0,C 180,E1 -4509.137,E2 -4509.137} C_VEL
LIN {X 0,Y 530.958,Z 222.352,A -85,B 0,C 180,E1 -4511.626,E2 -4511.626} C_VEL
LIN {X 0,Y 530.782,Z 222.374,A -85,B 0,C 180,E1 -4513.007,E2 -4513.007} C_VEL
LIN {X 0,Y 530.777,Z 223.794,A -85,B 0,C 180,E1 -4514.569,E2 -4514.569} C_VEL
LIN {X 0,Y 530.72,Z 227.341,A -85,B 0,C 180,E1 -4517.731,E2 -4517.731} C_VEL
LIN {X 0,Y 530.657,Z 230.025,A -85,B 0,C 180,E1 -4520.14,E2 -4520.14} C_VEL
LIN {X 0,Y 530.608,Z 233.575,A -85,B 0,C 180,E1 -4523.411,E2 -4523.411} C_VEL
LIN {X 0,Y 530.568,Z 236.427,A -85,B 0,C 180,E1 -4525.919,E2 -4525.919} C_VEL
LIN {X 0,Y 530.495,Z 239.266,A -85,B 0,C 180,E1 -4528.483,E2 -4528.483} C_VEL
LIN {X 0,Y 530.458,Z 242.194,A -85,B 0,C 180,E1 -4531.11,E2 -4531.11} C_VEL
LIN {X 0,Y 530.465,Z 244.969,A -85,B 0,C 180,E1 -4533.582,E2 -4533.582} C_VEL
LIN {X 0,Y 532.33,Z 255.449,A -85,B 0,C 180,E1 -4533.902,E2 -4533.902} C_VEL
LIN {X 0,Y 532.111,Z 268.452,A -85,B 0,C 180,E1 -4534.375,E2 -4534.375} C_VEL
LIN {X 0,Y 531.811,Z 280.678,A -85,B 0,C 180,E1 -4534.982,E2 -4534.982} C_VEL
LIN {X 0,Y 531.555,Z 291.479,A -85,B 0,C 180,E1 -4535.681,E2 -4535.681} C_VEL
LIN {X 0,Y 531.339,Z 301.904,A -85,B 0,C 180,E1 -4536.526,E2 -4536.526} C_VEL
LIN {X 0,Y 531.119,Z 311.582,A -85,B 0,C 180,E1 -4537.493,E2 -4537.493} C_VEL
LIN {X 0,Y 530.891,Z 319.617,A -85,B 0,C 180,E1 -4538.474,E2 -4538.474} C_VEL
LIN {X 0,Y 530.878,Z 320.941,A -85,B 0,C 180,E1 -4538.659,E2 -4538.659} C_VEL
LIN {X 0,Y 530.093,Z 324.515,A -85,B 0,C 180,E1 -4539.166,E2 -4539.166} C_VEL
LIN {X 0,Y 527.102,Z 329.942,A -85,B 0,C 180,E1 -4540.008,E2 -4540.008} C_VEL
LIN {X 0,Y 524.181,Z 334.695,A -85,B 0,C 180,E1 -4540.9,E2 -4540.9} C_VEL
LIN {X 0,Y 523.508,Z 337.195,A -85,B 0,C 180,E1 -4541.478,E2 -4541.478} C_VEL
LIN {X 0,Y 523.442,Z 341.712,A -85,B 0,C 180,E1 -4542.775,E2 -4542.775} C_VEL
LIN {X 0,Y 523.347,Z 345.297,A -85,B 0,C 180,E1 -4544.289,E2 -4544.289} C_VEL
LIN {X 0,Y 523.318,Z 347.236,A -85,B 0,C 180,E1 -4545.707,E2 -4545.707} C_VEL
LIN {X 0,Y 523.257,Z 347.787,A -85,B 0,C 180,E1 -4546.766,E2 -4546.766} C_VEL
LIN {X 0,Y 523.289,Z 347.617,A -85,B 0,C 180,E1 -4547.816,E2 -4547.816} C_VEL
LIN {X 0,Y 523.314,Z 346.743,A -85,B 0,C 180,E1 -4548.849,E2 -4548.849} C_VEL
LIN {X 0,Y 523.342,Z 344.021,A -85,B 0,C 180,E1 -4550.407,E2 -4550.407} C_VEL
LIN {X 0,Y 523.438,Z 339.953,A -85,B 0,C 180,E1 -4551.858,E2 -4551.858} C_VEL
LIN {X 0,Y 523.535,Z 334.335,A -85,B 0,C 180,E1 -4553.271,E2 -4553.271} C_VEL
LIN {X 0,Y 523.682,Z 327.86,A -85,B 0,C 180,E1 -4554.52,E2 -4554.52} C_VEL
LIN {X 0,Y 523.888,Z 320.122,A -85,B 0,C 180,E1 -4555.707,E2 -4555.707} C_VEL
LIN {X 0,Y 524.118,Z 311.543,A -85,B 0,C 180,E1 -4556.764,E2 -4556.764} C_VEL
LIN {X 0,Y 524.342,Z 302.424,A -85,B 0,C 180,E1 -4557.684,E2 -4557.684} C_VEL
LIN {X 0,Y 524.602,Z 292.517,A -85,B 0,C 180,E1 -4558.502,E2 -4558.502} C_VEL
LIN {X 0,Y 524.899,Z 280.934,A -85,B 0,C 180,E1 -4559.268,E2 -4559.268} C_VEL
LIN {X 0,Y 525.187,Z 268.774,A -85,B 0,C 180,E1 -4559.88,E2 -4559.88} C_VEL
LIN {X 0,Y 525.393,Z 255.324,A -85,B 0,C 180,E1 -4560.375,E2 -4560.375} C_VEL
LIN {X 0,Y 523.383,Z 245.146,A -85,B 0,C 180,E1 -4560.694,E2 -4560.694} C_VEL
LIN {X 0,Y 523.455,Z 241.224,A -85,B 0,C 180,E1 -4564.095,E2 -4564.095} C_VEL
LIN {X 0,Y 523.462,Z 237.794,A -85,B 0,C 180,E1 -4567.086,E2 -4567.086} C_VEL
LIN {X 0,Y 523.504,Z 234.017,A -85,B 0,C 180,E1 -4570.39,E2 -4570.39} C_VEL
LIN {X 0,Y 523.543,Z 231.282,A -85,B 0,C 180,E1 -4572.823,E2 -4572.823} C_VEL
LIN {X 0,Y 523.599,Z 228.535,A -85,B 0,C 180,E1 -4575.225,E2 -4575.225} C_VEL
LIN {X 0,Y 523.672,Z 224.924,A -85,B 0,C 180,E1 -4578.426,E2 -4578.426} C_VEL
LIN {X 0,Y 523.606,Z 223.266,A -85,B 0,C 180,E1 -4579.952,E2 -4579.952} C_VEL
LIN {X 0,Y 523.928,Z 223.225,A -85,B 0,C 180,E1 -4582.292,E2 -4582.292} C_VEL
LIN {X 0,Y 524.085,Z 223.205,A -85,B 0,C 180,E1 -4584.614,E2 -4584.614} C_VEL
LIN {X 0,Y 524.097,Z 223.202,A -85,B 0,C 180,E1 -4587.695,E2 -4587.695} C_VEL
LIN {X 0,Y 524.113,Z 223.203,A -85,B 0,C 180,E1 -4590.769,E2 -4590.769} C_VEL
LIN {X 0,Y 524.06,Z 223.21,A -85,B 0,C 180,E1 -4593.075,E2 -4593.075} C_VEL
LIN {X 0,Y 524.032,Z 223.21,A -85,B 0,C 180,E1 -4596.16,E2 -4596.16} C_VEL
LIN {X 0,Y 523.989,Z 223.217,A -85,B 0,C 180,E1 -4599.262,E2 -4599.262} C_VEL
LIN {X 0,Y 524.008,Z 223.213,A -85,B 0,C 180,E1 -4601.752,E2 -4601.752} C_VEL
LIN {X 0,Y 523.977,Z 223.219,A -85,B 0,C 180,E1 -4605.053,E2 -4605.053} C_VEL
LIN {X 0,Y 523.95,Z 223.219,A -85,B 0,C 180,E1 -4607.97,E2 -4607.97} C_VEL
LIN {X 0,Y 523.959,Z 223.219,A -85,B 0,C 180,E1 -4610.411,E2 -4610.411} C_VEL
LIN {X 0,Y 523.937,Z 223.223,A -85,B 0,C 180,E1 -4612.893,E2 -4612.893} C_VEL
LIN {X 0,Y 523.973,Z 223.218,A -85,B 0,C 180,E1 -4616.022,E2 -4616.022} C_VEL
LIN {X 0,Y 523.928,Z 223.224,A -85,B 0,C 180,E1 -4618.876,E2 -4618.876} C_VEL
LIN {X 0,Y 523.919,Z 223.226,A -85,B 0,C 180,E1 -4621.545,E2 -4621.545} C_VEL
LIN {X 0,Y 523.934,Z 223.224,A -85,B 0,C 180,E1 -4624.29,E2 -4624.29} C_VEL
LIN {X 0,Y 523.9,Z 223.227,A -85,B 0,C 180,E1 -4627.133,E2 -4627.133} C_VEL
LIN {X 0,Y 523.957,Z 223.222,A -85,B 0,C 180,E1 -4630.135,E2 -4630.135} C_VEL
LIN {X 0,Y 523.934,Z 223.225,A -85,B 0,C 180,E1 -4632.462,E2 -4632.462} C_VEL
LIN {X 0,Y 523.947,Z 223.22,A -85,B 0,C 180,E1 -4635.31,E2 -4635.31} C_VEL
LIN {X 0,Y 523.964,Z 223.219,A -85,B 0,C 180,E1 -4638.689,E2 -4638.689} C_VEL
LIN {X 0,Y 523.946,Z 223.22,A -85,B 0,C 180,E1 -4641.077,E2 -4641.077} C_VEL
LIN {X 0,Y 523.919,Z 223.224,A -85,B 0,C 180,E1 -4643.829,E2 -4643.829} C_VEL
LIN {X 0,Y 523.938,Z 223.225,A -85,B 0,C 180,E1 -4646.637,E2 -4646.637} C_VEL
LIN {X 0,Y 523.959,Z 223.22,A -85,B 0,C 180,E1 -4649.358,E2 -4649.358} C_VEL
LIN {X 0,Y 523.975,Z 223.218,A -85,B 0,C 180,E1 -4652.282,E2 -4652.282} C_VEL
LIN {X 0,Y 523.949,Z 223.221,A -85,B 0,C 180,E1 -4654.583,E2 -4654.583} C_VEL
LIN {X 0,Y 523.914,Z 223.226,A -85,B 0,C 180,E1 -4657.108,E2 -4657.108} C_VEL
LIN {X 0,Y 523.977,Z 223.22,A -85,B 0,C 180,E1 -4659.868,E2 -4659.868} C_VEL
LIN {X 0,Y 523.97,Z 223.218,A -85,B 0,C 180,E1 -4662.839,E2 -4662.839} C_VEL
LIN {X 0,Y 523.976,Z 223.216,A -85,B 0,C 180,E1 -4665.237,E2 -4665.237} C_VEL
LIN {X 0,Y 524.013,Z 223.213,A -85,B 0,C 180,E1 -4668.396,E2 -4668.396} C_VEL
LIN {X 0,Y 523.987,Z 223.217,A -85,B 0,C 180,E1 -4671.517,E2 -4671.517} C_VEL
LIN {X 0,Y 524.047,Z 223.21,A -85,B 0,C 180,E1 -4673.842,E2 -4673.842} C_VEL
LIN {X 0,Y 524.072,Z 223.205,A -85,B 0,C 180,E1 -4676.926,E2 -4676.926} C_VEL
LIN {X 0,Y 524.117,Z 223.203,A -85,B 0,C 180,E1 -4680.001,E2 -4680.001} C_VEL
LIN {X 0,Y 524.072,Z 223.205,A -85,B 0,C 180,E1 -4683.076,E2 -4683.076} C_VEL
LIN {X 0,Y 524.03,Z 223.211,A -85,B 0,C 180,E1 -4686.16,E2 -4686.16} C_VEL
LIN {X 0,Y 523.989,Z 223.216,A -85,B 0,C 180,E1 -4689.263,E2 -4689.263} C_VEL
LIN {X 0,Y 524.007,Z 223.215,A -85,B 0,C 180,E1 -4691.74,E2 -4691.74} C_VEL
LIN {X 0,Y 523.998,Z 223.214,A -85,B 0,C 180,E1 -4695.053,E2 -4695.053} C_VEL
LIN {X 0,Y 523.969,Z 223.219,A -85,B 0,C 180,E1 -4697.97,E2 -4697.97} C_VEL
LIN {X 0,Y 523.977,Z 223.218,A -85,B 0,C 180,E1 -4700.411,E2 -4700.411} C_VEL
LIN {X 0,Y 523.915,Z 223.227,A -85,B 0,C 180,E1 -4702.894,E2 -4702.894} C_VEL
LIN {X 0,Y 523.949,Z 223.222,A -85,B 0,C 180,E1 -4706.011,E2 -4706.011} C_VEL
LIN {X 0,Y 523.942,Z 223.223,A -85,B 0,C 180,E1 -4708.876,E2 -4708.876} C_VEL
LIN {X 0,Y 523.925,Z 223.224,A -85,B 0,C 180,E1 -4711.545,E2 -4711.545} C_VEL
LIN {X 0,Y 523.926,Z 223.224,A -85,B 0,C 180,E1 -4714.292,E2 -4714.292} C_VEL
LIN {X 0,Y 523.913,Z 223.227,A -85,B 0,C 180,E1 -4717.133,E2 -4717.133} C_VEL
LIN {X 0,Y 523.944,Z 223.221,A -85,B 0,C 180,E1 -4720.13,E2 -4720.13} C_VEL
LIN {X 0,Y 523.941,Z 223.221,A -85,B 0,C 180,E1 -4722.459,E2 -4722.459} C_VEL
LIN {X 0,Y 523.949,Z 223.222,A -85,B 0,C 180,E1 -4725.31,E2 -4725.31} C_VEL
LIN {X 0,Y 523.962,Z 223.221,A -85,B 0,C 180,E1 -4728.69,E2 -4728.69} C_VEL
LIN {X 0,Y 523.949,Z 223.357,A -85,B 0,C 180,E1 -4731.472,E2 -4731.472} C_VEL
LIN {X 0,Y 525.054,Z 229.698,A -85,B 0,C 180,E1 -4733.917,E2 -4733.917} C_VEL
LIN {X 0,Y 525.054,Z 235.944,A -85,B 0,C 180,E1 -4736.088,E2 -4736.088} C_VEL
LIN {X 0,Y 524.804,Z 244.519,A -85,B 0,C 180,E1 -4738.99,E2 -4738.99} C_VEL
LIN {X 0,Y 524.552,Z 254.082,A -85,B 0,C 180,E1 -4742.163,E2 -4742.163} C_VEL
LIN {X 0,Y 524.317,Z 262.956,A -85,B 0,C 180,E1 -4745.024,E2 -4745.024} C_VEL
LIN {X 0,Y 524.127,Z 272.224,A -85,B 0,C 180,E1 -4747.947,E2 -4747.947} C_VEL
LIN {X 0,Y 523.928,Z 281.491,A -85,B 0,C 180,E1 -4750.813,E2 -4750.813} C_VEL
LIN {X 0,Y 523.764,Z 290.758,A -85,B 0,C 180,E1 -4753.633,E2 -4753.633} C_VEL
LIN {X 0,Y 523.643,Z 299.709,A -85,B 0,C 180,E1 -4756.286,E2 -4756.286} C_VEL
LIN {X 0,Y 525.444,Z 311.254,A -85,B 0,C 180,E1 -4756.586,E2 -4756.586} C_VEL
LIN {X 0,Y 525.191,Z 323.761,A -85,B 0,C 180,E1 -4756.998,E2 -4756.998} C_VEL
LIN {X 0,Y 524.926,Z 335.404,A -85,B 0,C 180,E1 -4757.532,E2 -4757.532} C_VEL
LIN {X 0,Y 524.676,Z 346.663,A -85,B 0,C 180,E1 -4758.207,E2 -4758.207} C_VEL
LIN {X 0,Y 524.395,Z 358.257,A -85,B 0,C 180,E1 -4759.087,E2 -4759.087} C_VEL
LIN {X 0,Y 524.095,Z 367.535,A -85,B 0,C 180,E1 -4759.96,E2 -4759.96} C_VEL
LIN {X 0,Y 523.902,Z 375.988,A -85,B 0,C 180,E1 -4760.931,E2 -4760.931} C_VEL
LIN {X 0,Y 523.689,Z 384.235,A -85,B 0,C 180,E1 -4762.093,E2 -4762.093} C_VEL
LIN {X 0,Y 523.577,Z 389.866,A -85,B 0,C 180,E1 -4763.061,E2 -4763.061} C_VEL
LIN {X 0,Y 523.545,Z 395.364,A -85,B 0,C 180,E1 -4764.221,E2 -4764.221} C_VEL
LIN {X 0,Y 523.361,Z 399.676,A -85,B 0,C 180,E1 -4765.378,E2 -4765.378} C_VEL
LIN {X 0,Y 523.444,Z 401.956,A -85,B 0,C 180,E1 -4766.15,E2 -4766.15} C_VEL
LIN {X 0,Y 523.368,Z 403.807,A -85,B 0,C 180,E1 -4766.921,E2 -4766.921} C_VEL
LIN {X 0,Y 523.336,Z 405.196,A -85,B 0,C 180,E1 -4767.691,E2 -4767.691} C_VEL
LIN {X 0,Y 523.25,Z 406.785,A -85,B 0,C 180,E1 -4769.23,E2 -4769.23} C_VEL
LIN {X 0,Y 523.246,Z 407,A -85,B 0,C 180,E1 -4770,E2 -4770} C_VEL
LIN {X 0,Y 523.275,Z 406.186,A -85,B 0,C 180,E1 -4771.539,E2 -4771.539} C_VEL
LIN {X 0,Y 523.335,Z 405.199,A -85,B 0,C 180,E1 -4772.309,E2 -4772.309} C_VEL
LIN {X 0,Y 523.368,Z 403.811,A -85,B 0,C 180,E1 -4773.079,E2 -4773.079} C_VEL
LIN {X 0,Y 523.442,Z 400.897,A -85,B 0,C 180,E1 -4774.234,E2 -4774.234} C_VEL
LIN {X 0,Y 523.464,Z 396.95,A -85,B 0,C 180,E1 -4775.392,E2 -4775.392} C_VEL
LIN {X 0,Y 523.524,Z 391.734,A -85,B 0,C 180,E1 -4776.579,E2 -4776.579} C_VEL
LIN {X 0,Y 523.666,Z 385.471,A -85,B 0,C 180,E1 -4777.712,E2 -4777.712} C_VEL
LIN {X 0,Y 523.857,Z 377.482,A -85,B 0,C 180,E1 -4778.875,E2 -4778.875} C_VEL
LIN {X 0,Y 524.087,Z 369.34,A -85,B 0,C 180,E1 -4779.844,E2 -4779.844} C_VEL
LIN {X 0,Y 524.35,Z 359.406,A -85,B 0,C 180,E1 -4780.815,E2 -4780.815} C_VEL
LIN {X 0,Y 524.65,Z 348.26,A -85,B 0,C 180,E1 -4781.684,E2 -4781.684} C_VEL
LIN {X 0,Y 524.853,Z 337.185,A -85,B 0,C 180,E1 -4782.371,E2 -4782.371} C_VEL
LIN {X 0,Y 525.153,Z 324.99,A -85,B 0,C 180,E1 -4782.953,E2 -4782.953} C_VEL
LIN {X 0,Y 525.381,Z 312.194,A -85,B 0,C 180,E1 -4783.39,E2 -4783.39} C_VEL
LIN {X 0,Y 524.995,Z 307.942,A -85,B 0,C 180,E1 -4783.514,E2 -4783.514} C_VEL
LIN {X 0,Y 523.631,Z 299.532,A -85,B 0,C 180,E1 -4783.732,E2 -4783.732} C_VEL
LIN {X 0,Y 523.763,Z 290.761,A -85,B 0,C 180,E1 -4786.366,E2 -4786.366} C_VEL
LIN {X 0,Y 523.926,Z 281.494,A -85,B 0,C 180,E1 -4789.186,E2 -4789.186} C_VEL
LIN {X 0,Y 524.129,Z 271.44,A -85,B 0,C 180,E1 -4792.298,E2 -4792.298} C_VEL
LIN {X 0,Y 524.352,Z 261.635,A -85,B 0,C 180,E1 -4795.397,E2 -4795.397} C_VEL
LIN {X 0,Y 524.606,Z 252.368,A -85,B 0,C 180,E1 -4798.397,E2 -4798.397} C_VEL
LIN {X 0,Y 524.816,Z 242.96,A -85,B 0,C 180,E1 -4801.483,E2 -4801.483} C_VEL
LIN {X 0,Y 525.082,Z 233.512,A -85,B 0,C 180,E1 -4804.669,E2 -4804.669} C_VEL
LIN {X 0,Y 525.033,Z 229.583,A -85,B 0,C 180,E1 -4806.084,E2 -4806.084} C_VEL
LIN {X 0,Y 523.934,Z 223.225,A -85,B 0,C 180,E1 -4808.589,E2 -4808.589} C_VEL
LIN {X 0,Y 523.957,Z 223.223,A -85,B 0,C 180,E1 -4811.309,E2 -4811.309} C_VEL
LIN {X 0,Y 523.957,Z 223.222,A -85,B 0,C 180,E1 -4814.69,E2 -4814.69} C_VEL
LIN {X 0,Y 523.958,Z 223.221,A -85,B 0,C 180,E1 -4817.881,E2 -4817.881} C_VEL
LIN {X 0,Y 523.961,Z 223.222,A -85,B 0,C 180,E1 -4820.918,E2 -4820.918} C_VEL
LIN {X 0,Y 523.9,Z 223.229,A -85,B 0,C 180,E1 -4823.824,E2 -4823.824} C_VEL
LIN {X 0,Y 523.941,Z 223.223,A -85,B 0,C 180,E1 -4826.635,E2 -4826.635} C_VEL
LIN {X 0,Y 523.955,Z 223.221,A -85,B 0,C 180,E1 -4829.355,E2 -4829.355} C_VEL
LIN {X 0,Y 523.98,Z 223.219,A -85,B 0,C 180,E1 -4832.28,E2 -4832.28} C_VEL
LIN {X 0,Y 523.955,Z 223.221,A -85,B 0,C 180,E1 -4834.58,E2 -4834.58} C_VEL
LIN {X 0,Y 523.916,Z 223.225,A -85,B 0,C 180,E1 -4837.106,E2 -4837.106} C_VEL
LIN {X 0,Y 523.978,Z 223.217,A -85,B 0,C 180,E1 -4839.865,E2 -4839.865} C_VEL
LIN {X 0,Y 523.966,Z 223.22,A -85,B 0,C 180,E1 -4842.836,E2 -4842.836} C_VEL
LIN {X 0,Y 523.975,Z 223.218,A -85,B 0,C 180,E1 -4845.235,E2 -4845.235} C_VEL
LIN {X 0,Y 524.01,Z 223.214,A -85,B 0,C 180,E1 -4848.393,E2 -4848.393} C_VEL
LIN {X 0,Y 524.002,Z 223.214,A -85,B 0,C 180,E1 -4851.515,E2 -4851.515} C_VEL
LIN {X 0,Y 524.082,Z 223.205,A -85,B 0,C 180,E1 -4854.612,E2 -4854.612} C_VEL
LIN {X 0,Y 524.108,Z 223.201,A -85,B 0,C 180,E1 -4857.693,E2 -4857.693} C_VEL
LIN {X 0,Y 524.122,Z 223.2,A -85,B 0,C 180,E1 -4860.767,E2 -4860.767} C_VEL
LIN {X 0,Y 524.069,Z 223.207,A -85,B 0,C 180,E1 -4863.074,E2 -4863.074} C_VEL
LIN {X 0,Y 524.041,Z 223.211,A -85,B 0,C 180,E1 -4866.158,E2 -4866.158} C_VEL
LIN {X 0,Y 523.998,Z 223.216,A -85,B 0,C 180,E1 -4869.26,E2 -4869.26} C_VEL
LIN {X 0,Y 523.913,Z 223.23,A -85,B 0,C 180,E1 -4871.695,E2 -4871.695} C_VEL
LIN {X 0,Y 523.706,Z 223.255,A -85,B 0,C 180,E1 -4873.186,E2 -4873.186} C_VEL
LIN {X 0,Y 523.662,Z 225.668,A -85,B 0,C 180,E1 -4875.569,E2 -4875.569} C_VEL
LIN {X 0,Y 523.659,Z 228.347,A -85,B 0,C 180,E1 -4877.978,E2 -4877.978} C_VEL
LIN {X 0,Y 523.58,Z 231.04,A -85,B 0,C 180,E1 -4880.424,E2 -4880.424} C_VEL
LIN {X 0,Y 523.542,Z 233.795,A -85,B 0,C 180,E1 -4882.909,E2 -4882.909} C_VEL
LIN {X 0,Y 523.508,Z 237.079,A -85,B 0,C 180,E1 -4885.914,E2 -4885.914} C_VEL
LIN {X 0,Y 523.412,Z 240.421,A -85,B 0,C 180,E1 -4888.905,E2 -4888.905} C_VEL
LIN {X 0,Y 523.387,Z 243.408,A -85,B 0,C 180,E1 -4891.578,E2 -4891.578} C_VEL
LIN {X 0,Y 523.406,Z 245.451,A -85,B 0,C 180,E1 -4893.401,E2 -4893.401} C_VEL
LIN {X 0,Y 525.412,Z 255.687,A -85,B 0,C 180,E1 -4893.722,E2 -4893.722} C_VEL
LIN {X 0,Y 525.209,Z 268.541,A -85,B 0,C 180,E1 -4894.193,E2 -4894.193} C_VEL
LIN {X 0,Y 524.902,Z 280.649,A -85,B 0,C 180,E1 -4894.798,E2 -4894.798} C_VEL
LIN {X 0,Y 524.625,Z 291.649,A -85,B 0,C 180,E1 -4895.511,E2 -4895.511} C_VEL
LIN {X 0,Y 524.396,Z 301.374,A -85,B 0,C 180,E1 -4896.298,E2 -4896.298} C_VEL
LIN {X 0,Y 524.112,Z 311.038,A -85,B 0,C 180,E1 -4897.258,E2 -4897.258} C_VEL
LIN {X 0,Y 523.876,Z 319.613,A -85,B 0,C 180,E1 -4898.302,E2 -4898.302} C_VEL
LIN {X 0,Y 523.733,Z 326.594,A -85,B 0,C 180,E1 -4899.342,E2 -4899.342} C_VEL
LIN {X 0,Y 523.549,Z 333.468,A -85,B 0,C 180,E1 -4900.619,E2 -4900.619} C_VEL
LIN {X 0,Y 523.508,Z 337.195,A -85,B 0,C 180,E1 -4901.478,E2 -4901.478} C_VEL
LIN {X 0,Y 522.828,Z 339.492,A -85,B 0,C 180,E1 -4902.07,E2 -4902.07} C_VEL
LIN {X 0,Y 519.888,Z 342.753,A -85,B 0,C 180,E1 -4903.048,E2 -4903.048} C_VEL
LIN {X 0,Y 516.935,Z 345.34,A -85,B 0,C 180,E1 -4904.061,E2 -4904.061} C_VEL
LIN {X 0,Y 516.245,Z 346.43,A -85,B 0,C 180,E1 -4904.701,E2 -4904.701} C_VEL
LIN {X 0,Y 516.214,Z 348.008,A -85,B 0,C 180,E1 -4906.181,E2 -4906.181} C_VEL
LIN {X 0,Y 516.174,Z 348.216,A -85,B 0,C 180,E1 -4907.325,E2 -4907.325} C_VEL
LIN {X 0,Y 516.22,Z 347.57,A -85,B 0,C 180,E1 -4908.483,E2 -4908.483} C_VEL
LIN {X 0,Y 516.254,Z 346.006,A -85,B 0,C 180,E1 -4909.669,E2 -4909.669} C_VEL
LIN {X 0,Y 516.317,Z 343.424,A -85,B 0,C 180,E1 -4910.881,E2 -4910.881} C_VEL
LIN {X 0,Y 516.385,Z 339.277,A -85,B 0,C 180,E1 -4912.234,E2 -4912.234} C_VEL
LIN {X 0,Y 516.504,Z 334.56,A -85,B 0,C 180,E1 -4913.395,E2 -4913.395} C_VEL
LIN {X 0,Y 516.653,Z 327.815,A -85,B 0,C 180,E1 -4914.7,E2 -4914.7} C_VEL
LIN {X 0,Y 516.904,Z 320.178,A -85,B 0,C 180,E1 -4915.87,E2 -4915.87} C_VEL
LIN {X 0,Y 517.132,Z 311.4,A -85,B 0,C 180,E1 -4916.955,E2 -4916.955} C_VEL
LIN {X 0,Y 517.419,Z 301.892,A -85,B 0,C 180,E1 -4917.912,E2 -4917.912} C_VEL
LIN {X 0,Y 517.718,Z 291.247,A -85,B 0,C 180,E1 -4918.78,E2 -4918.78} C_VEL
LIN {X 0,Y 518.009,Z 279.531,A -85,B 0,C 180,E1 -4919.531,E2 -4919.531} C_VEL
